LIN {X 0,Y 112.861,Z 852.907,A -85,B 0,C 180,E1 29250,E2 29250} C_VEL
LIN {X 0,Y 107.228,Z 852.568,A -85,B 0,C 180,E1 29258.656,E2 29258.656} C_VEL
LIN {X 0,Y 96.977,Z 851.298,A -85,B 0,C 180,E1 29270.448,E2 29270.448} C_VEL
LIN {X 0,Y 87.732,Z 849.973,A -85,B 0,C 180,E1 29281.18,E2 29281.18} C_VEL
LIN {X 0,Y 77.61,Z 847.953,A -85,B 0,C 180,E1 29299.217,E2 29299.217} C_VEL
LIN {X 0,Y 60.63,Z 851.717,A -85,B 0,C 180,E1 29291.445,E2 29291.445} C_VEL
LIN {X 0,Y 43.178,Z 854.592,A -85,B 0,C 180,E1 29270.527,E2 29270.527} C_VEL
LIN {X 0,Y 38.153,Z 855.115,A -85,B 0,C 180,E1 29250,E2 29250} C_VEL
LIN {X 0,Y 52.851,Z 853.16,A -85,B 0,C 180,E1 29215.044,E2 29215.044} C_VEL
LIN {X 0,Y 73.881,Z 848.759,A -85,B 0,C 180,E1 29201.493,E2 29201.493} C_VEL
LIN {X 0,Y 77.759,Z 847.956,A -85,B 0,C 180,E1 29200.969,E2 29200.969} C_VEL
LIN {X 0,Y 88.144,Z 850.008,A -85,B 0,C 180,E1 29219.219,E2 29219.219} C_VEL
LIN {X 0,Y 99.484,Z 851.624,A -85,B 0,C 180,E1 29232.279,E2 29232.279} C_VEL
LIN {X 0,Y 103.001,Z 852.093,A -85,B 0,C 180,E1 29236.946,E2 29236.946} C_VEL
LIN {X 0,Y 106.169,Z 852.823,A -85,B 0,C 180,E1 29243.549,E2 29243.549} C_VEL
LIN {X 0,Y 104.929,Z 853.168,A -85,B 0,C 180,E1 29249.273,E2 29249.273} C_VEL
LIN {X 0,Y 104.315,Z 853.157,A -85,B 0,C 180,E1 29250.038,E2 29250.038} C_VEL
LIN {X 0,Y 97.922,Z 852.917,A -85,B 0,C 180,E1 29258.895,E2 29258.895} C_VEL
LIN {X 0,Y 87.911,Z 851.989,A -85,B 0,C 180,E1 29270.148,E2 29270.148} C_VEL
LIN {X 0,Y 73.225,Z 850.209,A -85,B 0,C 180,E1 29290.242,E2 29290.242} C_VEL
LIN {X 0,Y 50.776,Z 854.353,A -85,B 0,C 180,E1 29267.348,E2 29267.348} C_VEL
LIN {X 0,Y 46.131,Z 854.879,A -85,B 0,C 180,E1 29250,E2 29250} C_VEL
LIN {X 0,Y 59.659,Z 852.918,A -85,B 0,C 180,E1 29219.498,E2 29219.498} C_VEL
LIN {X 0,Y 73.337,Z 850.187,A -85,B 0,C 180,E1 29209.732,E2 29209.732} C_VEL
LIN {X 0,Y 87.957,Z 851.988,A -85,B 0,C 180,E1 29229.863,E2 29229.863} C_VEL
LIN {X 0,Y 97.92,Z 852.917,A -85,B 0,C 180,E1 29241.105,E2 29241.105} C_VEL
LIN {X 0,Y 104.315,Z 853.157,A -85,B 0,C 180,E1 29250.038,E2 29250.038} C_VEL
LIN {X 0,Y 96.304,Z 853.179,A -85,B 0,C 180,E1 29256,E2 29256} C_VEL
LIN {X 0,Y 81.253,Z 852.795,A -85,B 0,C 180,E1 29266.922,E2 29266.922} C_VEL
LIN {X 0,Y 70.197,Z 851.958,A -85,B 0,C 180,E1 29280.333,E2 29280.333} C_VEL
LIN {X 0,Y 54.121,Z 854.643,A -85,B 0,C 180,E1 29250,E2 29250} C_VEL
LIN {X 0,Y 70.111,Z 851.984,A -85,B 0,C 180,E1 29219.787,E2 29219.787} C_VEL
LIN {X 0,Y 79.937,Z 852.696,A -85,B 0,C 180,E1 29231.322,E2 29231.322} C_VEL
LIN {X 0,Y 88.018,Z 853.216,A -85,B 0,C 180,E1 29240.095,E2 29240.095} C_VEL
LIN {X 0,Y 95.517,Z 853.419,A -85,B 0,C 180,E1 29250,E2 29250} C_VEL
LIN {X 0,Y 88.015,Z 853.216,A -85,B 0,C 180,E1 29259.905,E2 29259.905} C_VEL
LIN {X 0,Y 81.253,Z 852.795,A -85,B 0,C 180,E1 29266.922,E2 29266.922} C_VEL
LIN {X 0,Y 76.697,Z 852.983,A -85,B 0,C 180,E1 29267.815,E2 29267.815} C_VEL
LIN {X 0,Y 68.723,Z 853.725,A -85,B 0,C 180,E1 29263.696,E2 29263.696} C_VEL
LIN {X 0,Y 63.261,Z 854.209,A -85,B 0,C 180,E1 29255.087,E2 29255.087} C_VEL
LIN {X 0,Y 62.099,Z 854.407,A -85,B 0,C 180,E1 29250,E2 29250} C_VEL
LIN {X 0,Y 67.517,Z 853.655,A -85,B 0,C 180,E1 29234.618,E2 29234.618} C_VEL
LIN {X 0,Y 70.634,Z 853.256,A -85,B 0,C 180,E1 29231.795,E2 29231.795} C_VEL
LIN {X 0,Y 81.708,Z 853.612,A -85,B 0,C 180,E1 29243.461,E2 29243.461} C_VEL
LIN {X 0,Y 86.693,Z 853.68,A -85,B 0,C 180,E1 29250,E2 29250} C_VEL
LIN {X 0,Y 81.704,Z 853.612,A -85,B 0,C 180,E1 29256.541,E2 29256.541} C_VEL
LIN {X 0,Y 70.562,Z 853.261,A -85,B 0,C 180,E1 29268.197,E2 29268.197} C_VEL
LIN {X 0,Y 66.314,Z 853.874,A -85,B 0,C 180,E1 29263.198,E2 29263.198} C_VEL
LIN {X 0,Y 63.261,Z 854.209,A -85,B 0,C 180,E1 29255.087,E2 29255.087} C_VEL
LIN {X 0,Y 64.956,Z 854.291,A -85,B 0,C 180,E1 29248.536,E2 29248.536} C_VEL
LIN {X 0,Y 70.805,Z 854.008,A -85,B 0,C 180,E1 29244.483,E2 29244.483} C_VEL
LIN {X 0,Y 73.194,Z 853.938,A -85,B 0,C 180,E1 29244.98,E2 29244.98} C_VEL
LIN {X 0,Y 77.516,Z 853.951,A -85,B 0,C 180,E1 29250,E2 29250} C_VEL
LIN {X 0,Y 73.194,Z 853.938,A -85,B 0,C 180,E1 29255.016,E2 29255.016} C_VEL
LIN {X 0,Y 70.1,Z 854.17,A -85,B 0,C 180,E1 29250,E2 29250} C_VEL
LIN {X 0,Y 73.194,Z 853.938,A -85,B 0,C 180,E1 29244.98,E2 29244.98} C_VEL
LIN {X 0,Y 74.21,Z 855.937,A -85,B 0,C 180,E1 29243.58,E2 29243.58} C_VEL
LIN {X 0,Y 74.21,Z 875,A -85,B 0,C 180,E1 29243.58,E2 29243.58} C_VEL
LIN {X 0,Y 74.21,Z 875,A -85,B 0,C 180,E1 29243.58,E2 29243.58}

QRS_NEXT_CUT()
PTP {E1 29336.94,E2 29336.94}
PTP {X 0,Y 607.852,A -85,B 0,C 180,E1 29336.94,E2 29336.94,E3 0,E4 0,E5 0,E6 0}
QRS_SPEED_INIT()
LIN {X 0,Y 607.852,Z 875,A -85,B 0,C 180,E1 29336.94,E2 29336.94,E3 0,E4 0,E5 0,E6 0} C_VEL
LIN {X 0,Y 607.852,Z 359.34,A -85,B 0,C 180,E1 29336.94,E2 29336.94} C_VEL
LIN {X 0,Y 607.852,Z 351.263,A -85,B 0,C 180,E1 29336.94,E2 29336.94} C_VEL
LIN {X 0,Y 607.872,Z 349.263,A -85,B 0,C 180,E1 29336.752,E2 29336.752} C_VEL
LIN {X 0,Y 607.835,Z 349.264,A -85,B 0,C 180,E1 29333.582,E2 29333.582} C_VEL
LIN {X 0,Y 607.853,Z 349.263,A -85,B 0,C 180,E1 29330.824,E2 29330.824} C_VEL
LIN {X 0,Y 607.845,Z 349.264,A -85,B 0,C 180,E1 29327.658,E2 29327.658} C_VEL
LIN {X 0,Y 607.838,Z 349.264,A -85,B 0,C 180,E1 29324.918,E2 29324.918} C_VEL
LIN {X 0,Y 607.857,Z 349.264,A -85,B 0,C 180,E1 29321.695,E2 29321.695} C_VEL
LIN {X 0,Y 607.831,Z 349.264,A -85,B 0,C 180,E1 29318.992,E2 29318.992} C_VEL
LIN {X 0,Y 607.895,Z 349.264,A -85,B 0,C 180,E1 29315.899,E2 29315.899} C_VEL
LIN {X 0,Y 607.83,Z 349.264,A -85,B 0,C 180,E1 29312.9,E2 29312.9} C_VEL
LIN {X 0,Y 607.892,Z 349.265,A -85,B 0,C 180,E1 29309.788,E2 29309.788} C_VEL
LIN {X 0,Y 607.829,Z 349.264,A -85,B 0,C 180,E1 29306.852,E2 29306.852} C_VEL
LIN {X 0,Y 607.91,Z 349.265,A -85,B 0,C 180,E1 29303.818,E2 29303.818} C_VEL
LIN {X 0,Y 607.828,Z 349.264,A -85,B 0,C 180,E1 29300.835,E2 29300.835} C_VEL
LIN {X 0,Y 607.916,Z 349.265,A -85,B 0,C 180,E1 29297.734,E2 29297.734} C_VEL
LIN {X 0,Y 607.828,Z 349.265,A -85,B 0,C 180,E1 29294.724,E2 29294.724} C_VEL
LIN {X 0,Y 607.914,Z 349.265,A -85,B 0,C 180,E1 29291.705,E2 29291.705} C_VEL
LIN {X 0,Y 607.827,Z 349.265,A -85,B 0,C 180,E1 29288.626,E2 29288.626} C_VEL
LIN {X 0,Y 607.912,Z 349.265,A -85,B 0,C 180,E1 29285.607,E2 29285.607} C_VEL
LIN {X 0,Y 607.828,Z 349.265,A -85,B 0,C 180,E1 29282.638,E2 29282.638} C_VEL
LIN {X 0,Y 607.88,Z 349.264,A -85,B 0,C 180,E1 29279.734,E2 29279.734} C_VEL
LIN {X 0,Y 607.832,Z 349.265,A -85,B 0,C 180,E1 29276.683,E2 29276.683} C_VEL
LIN {X 0,Y 607.852,Z 349.265,A -85,B 0,C 180,E1 29273.868,E2 29273.868} C_VEL
LIN {X 0,Y 607.834,Z 349.265,A -85,B 0,C 180,E1 29270.636,E2 29270.636} C_VEL
LIN {X 0,Y 607.839,Z 349.265,A -85,B 0,C 180,E1 29267.914,E2 29267.914} C_VEL
LIN {X 0,Y 607.836,Z 349.265,A -85,B 0,C 180,E1 29264.576,E2 29264.576} C_VEL
LIN {X 0,Y 607.835,Z 349.265,A -85,B 0,C 180,E1 29261.865,E2 29261.865} C_VEL
LIN {X 0,Y 607.846,Z 349.265,A -85,B 0,C 180,E1 29258.609,E2 29258.609} C_VEL
LIN {X 0,Y 607.827,Z 349.265,A -85,B 0,C 180,E1 29255.948,E2 29255.948} C_VEL
LIN {X 0,Y 607.897,Z 349.265,A -85,B 0,C 180,E1 29252.923,E2 29252.923} C_VEL
LIN {X 0,Y 607.825,Z 349.265,A -85,B 0,C 180,E1 29249.906,E2 29249.906} C_VEL
LIN {X 0,Y 607.9,Z 349.266,A -85,B 0,C 180,E1 29246.889,E2 29246.889} C_VEL
LIN {X 0,Y 607.825,Z 349.265,A -85,B 0,C 180,E1 29243.957,E2 29243.957} C_VEL
LIN {X 0,Y 607.893,Z 349.265,A -85,B 0,C 180,E1 29241.011,E2 29241.011} C_VEL
LIN {X 0,Y 607.827,Z 349.265,A -85,B 0,C 180,E1 29237.942,E2 29237.942} C_VEL
LIN {X 0,Y 607.875,Z 349.265,A -85,B 0,C 180,E1 29235.035,E2 29235.035} C_VEL
LIN {X 0,Y 607.83,Z 349.265,A -85,B 0,C 180,E1 29231.924,E2 29231.924} C_VEL
LIN {X 0,Y 607.857,Z 349.265,A -85,B 0,C 180,E1 29229.088,E2 29229.088} C_VEL
LIN {X 0,Y 607.834,Z 349.265,A -85,B 0,C 180,E1 29225.897,E2 29225.897} C_VEL
LIN {X 0,Y 607.846,Z 349.265,A -85,B 0,C 180,E1 29223.106,E2 29223.106} C_VEL
LIN {X 0,Y 607.84,Z 349.265,A -85,B 0,C 180,E1 29219.888,E2 29219.888} C_VEL
LIN {X 0,Y 607.838,Z 349.265,A -85,B 0,C 180,E1 29217.125,E2 29217.125} C_VEL
LIN {X 0,Y 607.842,Z 349.264,A -85,B 0,C 180,E1 29213.807,E2 29213.807} C_VEL
LIN {X 0,Y 607.835,Z 349.265,A -85,B 0,C 180,E1 29211.071,E2 29211.071} C_VEL
LIN {X 0,Y 607.855,Z 349.264,A -85,B 0,C 180,E1 29207.848,E2 29207.848} C_VEL
LIN {X 0,Y 607.83,Z 349.265,A -85,B 0,C 180,E1 29205.116,E2 29205.116} C_VEL
LIN {X 0,Y 607.902,Z 349.264,A -85,B 0,C 180,E1 29202.118,E2 29202.118} C_VEL
LIN {X 0,Y 607.829,Z 349.264,A -85,B 0,C 180,E1 29199.068,E2 29199.068} C_VEL
LIN {X 0,Y 607.913,Z 349.264,A -85,B 0,C 180,E1 29196.065,E2 29196.065} C_VEL
LIN {X 0,Y 607.829,Z 349.264,A -85,B 0,C 180,E1 29193.094,E2 29193.094} C_VEL
LIN {X 0,Y 607.908,Z 349.265,A -85,B 0,C 180,E1 29190.102,E2 29190.102} C_VEL
LIN {X 0,Y 607.83,Z 349.264,A -85,B 0,C 180,E1 29187.1,E2 29187.1} C_VEL
LIN {X 0,Y 607.9,Z 349.264,A -85,B 0,C 180,E1 29184.067,E2 29184.067} C_VEL
LIN {X 0,Y 607.831,Z 349.264,A -85,B 0,C 180,E1 29181.008,E2 29181.008} C_VEL
LIN {X 0,Y 607.867,Z 349.264,A -85,B 0,C 180,E1 29178.206,E2 29178.206} C_VEL
LIN {X 0,Y 607.836,Z 349.264,A -85,B 0,C 180,E1 29175.059,E2 29175.059} C_VEL
LIN {X 0,Y 607.845,Z 349.264,A -85,B 0,C 180,E1 29172.342,E2 29172.342} C_VEL
LIN {X 0,Y 607.845,Z 349.263,A -85,B 0,C 180,E1 29169.081,E2 29169.081} C_VEL
LIN {X 0,Y 607.835,Z 349.264,A -85,B 0,C 180,E1 29166.418,E2 29166.418} C_VEL
LIN {X 0,Y 607.872,Z 349.263,A -85,B 0,C 180,E1 29163.248,E2 29163.248} C_VEL
LIN {X 0,Y 607.833,Z 349.264,A -85,B 0,C 180,E1 29160.373,E2 29160.373} C_VEL
LIN {X 0,Y 607.888,Z 349.263,A -85,B 0,C 180,E1 29157.262,E2 29157.262} C_VEL
LIN {X 0,Y 607.833,Z 349.263,A -85,B 0,C 180,E1 29154.332,E2 29154.332} C_VEL
LIN {X 0,Y 607.904,Z 349.264,A -85,B 0,C 180,E1 29151.292,E2 29151.292} C_VEL
LIN {X 0,Y 607.832,Z 349.264,A -85,B 0,C 180,E1 29148.323,E2 29148.323} C_VEL
LIN {X 0,Y 607.915,Z 349.264,A -85,B 0,C 180,E1 29145.325,E2 29145.325} C_VEL
LIN {X 0,Y 607.832,Z 349.264,A -85,B 0,C 180,E1 29142.251,E2 29142.251} C_VEL
LIN {X 0,Y 607.909,Z 349.264,A -85,B 0,C 180,E1 29139.187,E2 29139.187} C_VEL
LIN {X 0,Y 607.833,Z 349.264,A -85,B 0,C 180,E1 29136.128,E2 29136.128} C_VEL
LIN {X 0,Y 607.911,Z 349.264,A -85,B 0,C 180,E1 29133.106,E2 29133.106} C_VEL
LIN {X 0,Y 607.834,Z 349.264,A -85,B 0,C 180,E1 29130.096,E2 29130.096} C_VEL
LIN {X 0,Y 607.907,Z 349.265,A -85,B 0,C 180,E1 29127.125,E2 29127.125} C_VEL
LIN {X 0,Y 607.838,Z 349.264,A -85,B 0,C 180,E1 29124.153,E2 29124.153} C_VEL
LIN {X 0,Y 607.861,Z 349.264,A -85,B 0,C 180,E1 29121.379,E2 29121.379} C_VEL
LIN {X 0,Y 607.844,Z 349.263,A -85,B 0,C 180,E1 29118.17,E2 29118.17} C_VEL
LIN {X 0,Y 607.852,Z 349.264,A -85,B 0,C 180,E1 29115.381,E2 29115.381} C_VEL
LIN {X 0,Y 607.846,Z 349.263,A -85,B 0,C 180,E1 29112.109,E2 29112.109} C_VEL
LIN {X 0,Y 607.847,Z 349.264,A -85,B 0,C 180,E1 29109.364,E2 29109.364} C_VEL
LIN {X 0,Y 607.852,Z 349.263,A -85,B 0,C 180,E1 29106.076,E2 29106.076} C_VEL
LIN {X 0,Y 607.844,Z 349.263,A -85,B 0,C 180,E1 29103.318,E2 29103.318} C_VEL
LIN {X 0,Y 607.896,Z 349.549,A -85,B 0,C 180,E1 29102.807,E2 29102.807} C_VEL
LIN {X 0,Y 607.904,Z 374.795,A -85,B 0,C 180,E1 29099.891,E2 29099.891} C_VEL
LIN {X 0,Y 607.881,Z 395.066,A -85,B 0,C 180,E1 29097.648,E2 29097.648} C_VEL
LIN {X 0,Y 607.918,Z 609.038,A -85,B 0,C 180,E1 29094.874,E2 29094.874} C_VEL
LIN {X 0,Y 607.917,Z 654.447,A -85,B 0,C 180,E1 29094.265,E2 29094.265} C_VEL
LIN {X 0,Y 607.906,Z 675.785,A -85,B 0,C 180,E1 29093.789,E2 29093.789} C_VEL
LIN {X 0,Y 607.91,Z 694.347,A -85,B 0,C 180,E1 29093.204,E2 29093.204} C_VEL
LIN {X 0,Y 607.913,Z 713.651,A -85,B 0,C 180,E1 29092.43,E2 29092.43} C_VEL
LIN {X 0,Y 607.919,Z 732.066,A -85,B 0,C 180,E1 29091.516,E2 29091.516} C_VEL
LIN {X 0,Y 607.917,Z 750.545,A -85,B 0,C 180,E1 29090.406,E2 29090.406} C_VEL
LIN {X 0,Y 607.912,Z 768.568,A -85,B 0,C 180,E1 29089.105,E2 29089.105} C_VEL
LIN {X 0,Y 607.916,Z 785.369,A -85,B 0,C 180,E1 29087.665,E2 29087.665} C_VEL
LIN {X 0,Y 607.909,Z 800.458,A -85,B 0,C 180,E1 29086.138,E2 29086.138} C_VEL
LIN {X 0,Y 607.911,Z 813.589,A -85,B 0,C 180,E1 29084.574,E2 29084.574} C_VEL
LIN {X 0,Y 607.917,Z 825.378,A -85,B 0,C 180,E1 29082.925,E2 29082.925} C_VEL
LIN {X 0,Y 607.912,Z 836.326,A -85,B 0,C 180,E1 29081.095,E2 29081.095} C_VEL
LIN {X 0,Y 607.917,Z 845.249,A -85,B 0,C 180,E1 29079.275,E2 29079.275} C_VEL
LIN {X 0,Y 607.914,Z 852.378,A -85,B 0,C 180,E1 29077.466,E2 29077.466} C_VEL
LIN {X 0,Y 607.912,Z 858.002,A -85,B 0,C 180,E1 29075.569,E2 29075.569} C_VEL
LIN {X 0,Y 607.911,Z 861.924,A -85,B 0,C 180,E1 29073.678,E2 29073.678} C_VEL
LIN {X 0,Y 607.907,Z 864.307,A -85,B 0,C 180,E1 29071.696,E2 29071.696} C_VEL
LIN {X 0,Y 607.907,Z 864.962,A -85,B 0,C 180,E1 29069.812,E2 29069.812} C_VEL
LIN {X 0,Y 607.909,Z 863.95,A -85,B 0,C 180,E1 29067.832,E2 29067.832} C_VEL
LIN {X 0,Y 607.909,Z 861.135,A -85,B 0,C 180,E1 29065.85,E2 29065.85} C_VEL
LIN {X 0,Y 607.916,Z 856.736,A -85,B 0,C 180,E1 29063.958,E2 29063.958} C_VEL
LIN {X 0,Y 607.905,Z 850.621,A -85,B 0,C 180,E1 29062.059,E2 29062.059} C_VEL
LIN {X 0,Y 607.903,Z 843.098,A -85,B 0,C 180,E1 29060.247,E2 29060.247} C_VEL
LIN {X 0,Y 607.904,Z 833.718,A -85,B 0,C 180,E1 29058.425,E2 29058.425} C_VEL
LIN {X 0,Y 607.915,Z 822.179,A -85,B 0,C 180,E1 29056.591,E2 29056.591} C_VEL
LIN {X 0,Y 607.917,Z 809.38,A -85,B 0,C 180,E1 29054.897,E2 29054.897} C_VEL
LIN {X 0,Y 607.911,Z 795.823,A -85,B 0,C 180,E1 29053.371,E2 29053.371} C_VEL
LIN {X 0,Y 607.912,Z 780.817,A -85,B 0,C 180,E1 29051.927,E2 29051.927} C_VEL
LIN {X 0,Y 607.916,Z 763.955,A -85,B 0,C 180,E1 29050.546,E2 29050.546} C_VEL
LIN {X 0,Y 607.918,Z 746.338,A -85,B 0,C 180,E1 29049.329,E2 29049.329} C_VEL
LIN {X 0,Y 607.918,Z 728.275,A -85,B 0,C 180,E1 29048.281,E2 29048.281} C_VEL
LIN {X 0,Y 607.918,Z 709.066,A -85,B 0,C 180,E1 29047.365,E2 29047.365} C_VEL
LIN {X 0,Y 607.916,Z 690.111,A -85,B 0,C 180,E1 29046.649,E2 29046.649} C_VEL
LIN {X 0,Y 607.907,Z 670.6,A -85,B 0,C 180,E1 29046.082,E2 29046.082} C_VEL
LIN {X 0,Y 607.917,Z 650.327,A -85,B 0,C 180,E1 29045.67,E2 29045.67} C_VEL
LIN {X 0,Y 607.884,Z 404.447,A -85,B 0,C 180,E1 29042.485,E2 29042.485} C_VEL
LIN {X 0,Y 607.881,Z 394.817,A -85,B 0,C 180,E1 29042.339,E2 29042.339} C_VEL
LIN {X 0,Y 607.916,Z 367.575,A -85,B 0,C 180,E1 29039.288,E2 29039.288} C_VEL
LIN {X 0,Y 607.891,Z 349.374,A -85,B 0,C 180,E1 29037.152,E2 29037.152} C_VEL
LIN {X 0,Y 607.836,Z 349.264,A -85,B 0,C 180,E1 29034.272,E2 29034.272} C_VEL
LIN {X 0,Y 607.913,Z 349.265,A -85,B 0,C 180,E1 29031.198,E2 29031.198} C_VEL
LIN {X 0,Y 607.835,Z 349.263,A -85,B 0,C 180,E1 29028.227,E2 29028.227} C_VEL
LIN {X 0,Y 607.914,Z 349.263,A -85,B 0,C 180,E1 29025.257,E2 29025.257} C_VEL
LIN {X 0,Y 607.835,Z 349.264,A -85,B 0,C 180,E1 29022.251,E2 29022.251} C_VEL
LIN {X 0,Y 607.885,Z 349.263,A -85,B 0,C 180,E1 29019.372,E2 29019.372} C_VEL
LIN {X 0,Y 607.839,Z 349.264,A -85,B 0,C 180,E1 29016.294,E2 29016.294} C_VEL
LIN {X 0,Y 607.853,Z 349.263,A -85,B 0,C 180,E1 29013.554,E2 29013.554} C_VEL
LIN {X 0,Y 607.844,Z 349.264,A -85,B 0,C 180,E1 29010.281,E2 29010.281} C_VEL
LIN {X 0,Y 607.855,Z 349.262,A -85,B 0,C 180,E1 29007.426,E2 29007.426} C_VEL
LIN {X 0,Y 607.843,Z 349.264,A -85,B 0,C 180,E1 29004.182,E2 29004.182} C_VEL
LIN {X 0,Y 607.848,Z 349.263,A -85,B 0,C 180,E1 29001.41,E2 29001.41} C_VEL
LIN {X 0,Y 607.844,Z 349.264,A -85,B 0,C 180,E1 28998.116,E2 28998.116} C_VEL
LIN {X 0,Y 607.844,Z 349.263,A -85,B 0,C 180,E1 28995.36,E2 28995.36} C_VEL
LIN {X 0,Y 607.848,Z 349.264,A -85,B 0,C 180,E1 28992.061,E2 28992.061} C_VEL
LIN {X 0,Y 607.842,Z 349.264,A -85,B 0,C 180,E1 28989.28,E2 28989.28} C_VEL
LIN {X 0,Y 607.846,Z 349.264,A -85,B 0,C 180,E1 28985.952,E2 28985.952} C_VEL
LIN {X 0,Y 607.846,Z 349.264,A -85,B 0,C 180,E1 28983.116,E2 28983.116} C_VEL
LIN {X 0,Y 607.843,Z 349.264,A -85,B 0,C 180,E1 28979.816,E2 28979.816} C_VEL
LIN {X 0,Y 607.842,Z 349.263,A -85,B 0,C 180,E1 28977.081,E2 28977.081} C_VEL
LIN {X 0,Y 607.872,Z 349.263,A -85,B 0,C 180,E1 28976.752,E2 28976.752} C_VEL
LIN {X 0,Y 606.937,Z 349.386,A -85,B 0,C 180,E1 28976.025,E2 28976.025} C_VEL
LIN {X 0,Y 600.442,Z 350.191,A -85,B 0,C 180,E1 28973.989,E2 28973.989} C_VEL
LIN {X 0,Y 599.893,Z 350.253,A -85,B 0,C 180,E1 28973.458,E2 28973.458} C_VEL
LIN {X 0,Y 599.939,Z 350.25,A -85,B 0,C 180,E1 28970.605,E2 28970.605} C_VEL
LIN {X 0,Y 599.897,Z 350.253,A -85,B 0,C 180,E1 28967.491,E2 28967.491} C_VEL
LIN {X 0,Y 599.912,Z 350.253,A -85,B 0,C 180,E1 28964.737,E2 28964.737} C_VEL
LIN {X 0,Y 599.899,Z 350.253,A -85,B 0,C 180,E1 28961.443,E2 28961.443} C_VEL
LIN {X 0,Y 599.917,Z 350.253,A -85,B 0,C 180,E1 28958.599,E2 28958.599} C_VEL
LIN {X 0,Y 599.9,Z 350.252,A -85,B 0,C 180,E1 28955.382,E2 28955.382} C_VEL
LIN {X 0,Y 599.915,Z 350.253,A -85,B 0,C 180,E1 28952.512,E2 28952.512} C_VEL
LIN {X 0,Y 599.902,Z 350.254,A -85,B 0,C 180,E1 28949.316,E2 28949.316} C_VEL
LIN {X 0,Y 599.905,Z 350.253,A -85,B 0,C 180,E1 28946.526,E2 28946.526} C_VEL
LIN {X 0,Y 599.904,Z 350.254,A -85,B 0,C 180,E1 28943.257,E2 28943.257} C_VEL
LIN {X 0,Y 599.895,Z 350.253,A -85,B 0,C 180,E1 28940.587,E2 28940.587} C_VEL
LIN {X 0,Y 599.93,Z 350.254,A -85,B 0,C 180,E1 28937.427,E2 28937.427} C_VEL
LIN {X 0,Y 599.891,Z 350.254,A -85,B 0,C 180,E1 28934.561,E2 28934.561} C_VEL
LIN {X 0,Y 599.943,Z 350.254,A -85,B 0,C 180,E1 28931.423,E2 28931.423} C_VEL
LIN {X 0,Y 599.892,Z 350.254,A -85,B 0,C 180,E1 28928.438,E2 28928.438} C_VEL
LIN {X 0,Y 599.933,Z 350.254,A -85,B 0,C 180,E1 28925.263,E2 28925.263} C_VEL
LIN {X 0,Y 599.888,Z 350.254,A -85,B 0,C 180,E1 28922.458,E2 28922.458} C_VEL
LIN {X 0,Y 599.959,Z 350.255,A -85,B 0,C 180,E1 28919.37,E2 28919.37} C_VEL
LIN {X 0,Y 599.888,Z 350.254,A -85,B 0,C 180,E1 28916.424,E2 28916.424} C_VEL
LIN {X 0,Y 599.973,Z 350.254,A -85,B 0,C 180,E1 28913.349,E2 28913.349} C_VEL
LIN {X 0,Y 599.888,Z 350.254,A -85,B 0,C 180,E1 28910.386,E2 28910.386} C_VEL
LIN {X 0,Y 599.962,Z 350.255,A -85,B 0,C 180,E1 28907.356,E2 28907.356} C_VEL
LIN {X 0,Y 599.889,Z 350.254,A -85,B 0,C 180,E1 28904.379,E2 28904.379} C_VEL
LIN {X 0,Y 599.928,Z 350.254,A -85,B 0,C 180,E1 28901.526,E2 28901.526} C_VEL
LIN {X 0,Y 599.894,Z 350.254,A -85,B 0,C 180,E1 28898.434,E2 28898.434} C_VEL
LIN {X 0,Y 599.898,Z 350.254,A -85,B 0,C 180,E1 28895.739,E2 28895.739} C_VEL
LIN {X 0,Y 599.897,Z 350.254,A -85,B 0,C 180,E1 28892.388,E2 28892.388} C_VEL
LIN {X 0,Y 599.899,Z 350.254,A -85,B 0,C 180,E1 28889.618,E2 28889.618} C_VEL
LIN {X 0,Y 599.896,Z 350.254,A -85,B 0,C 180,E1 28886.273,E2 28886.273} C_VEL
LIN {X 0,Y 599.902,Z 350.254,A -85,B 0,C 180,E1 28883.493,E2 28883.493} C_VEL
LIN {X 0,Y 599.9,Z 350.254,A -85,B 0,C 180,E1 28880.212,E2 28880.212} C_VEL
LIN {X 0,Y 599.902,Z 350.254,A -85,B 0,C 180,E1 28877.389,E2 28877.389} C_VEL
LIN {X 0,Y 599.896,Z 350.254,A -85,B 0,C 180,E1 28874.061,E2 28874.061} C_VEL
LIN {X 0,Y 599.908,Z 350.254,A -85,B 0,C 180,E1 28871.237,E2 28871.237} C_VEL
LIN {X 0,Y 599.898,Z 350.254,A -85,B 0,C 180,E1 28867.976,E2 28867.976} C_VEL
LIN {X 0,Y 599.898,Z 350.254,A -85,B 0,C 180,E1 28865.261,E2 28865.261} C_VEL
LIN {X 0,Y 599.904,Z 350.254,A -85,B 0,C 180,E1 28861.966,E2 28861.966} C_VEL
LIN {X 0,Y 599.895,Z 350.254,A -85,B 0,C 180,E1 28859.225,E2 28859.225} C_VEL
LIN {X 0,Y 599.924,Z 350.254,A -85,B 0,C 180,E1 28856.061,E2 28856.061} C_VEL
LIN {X 0,Y 599.891,Z 350.254,A -85,B 0,C 180,E1 28853.249,E2 28853.249} C_VEL
LIN {X 0,Y 599.955,Z 350.253,A -85,B 0,C 180,E1 28850.188,E2 28850.188} C_VEL
LIN {X 0,Y 599.889,Z 350.254,A -85,B 0,C 180,E1 28847.286,E2 28847.286} C_VEL
LIN {X 0,Y 599.974,Z 350.254,A -85,B 0,C 180,E1 28844.228,E2 28844.228} C_VEL
LIN {X 0,Y 599.89,Z 350.254,A -85,B 0,C 180,E1 28841.264,E2 28841.264} C_VEL
LIN {X 0,Y 599.976,Z 350.253,A -85,B 0,C 180,E1 28838.135,E2 28838.135} C_VEL
LIN {X 0,Y 599.89,Z 350.254,A -85,B 0,C 180,E1 28835.081,E2 28835.081} C_VEL
LIN {X 0,Y 599.971,Z 350.253,A -85,B 0,C 180,E1 28831.995,E2 28831.995} C_VEL
LIN {X 0,Y 599.891,Z 350.253,A -85,B 0,C 180,E1 28828.954,E2 28828.954} C_VEL
LIN {X 0,Y 599.963,Z 350.252,A -85,B 0,C 180,E1 28825.855,E2 28825.855} C_VEL
LIN {X 0,Y 599.892,Z 350.252,A -85,B 0,C 180,E1 28822.828,E2 28822.828} C_VEL
LIN {X 0,Y 599.969,Z 350.252,A -85,B 0,C 180,E1 28819.768,E2 28819.768} C_VEL
LIN {X 0,Y 599.892,Z 350.251,A -85,B 0,C 180,E1 28816.753,E2 28816.753} C_VEL
LIN {X 0,Y 599.967,Z 350.253,A -85,B 0,C 180,E1 28813.683,E2 28813.683} C_VEL
LIN {X 0,Y 599.892,Z 350.252,A -85,B 0,C 180,E1 28810.657,E2 28810.657} C_VEL
LIN {X 0,Y 599.967,Z 350.252,A -85,B 0,C 180,E1 28807.561,E2 28807.561} C_VEL
LIN {X 0,Y 599.892,Z 350.253,A -85,B 0,C 180,E1 28804.584,E2 28804.584} C_VEL
LIN {X 0,Y 599.974,Z 350.251,A -85,B 0,C 180,E1 28801.524,E2 28801.524} C_VEL
LIN {X 0,Y 599.894,Z 350.253,A -85,B 0,C 180,E1 28798.468,E2 28798.468} C_VEL
LIN {X 0,Y 599.971,Z 350.251,A -85,B 0,C 180,E1 28795.408,E2 28795.408} C_VEL
LIN {X 0,Y 599.893,Z 350.251,A -85,B 0,C 180,E1 28792.43,E2 28792.43} C_VEL
LIN {X 0,Y 599.973,Z 350.253,A -85,B 0,C 180,E1 28789.336,E2 28789.336} C_VEL
LIN {X 0,Y 599.894,Z 350.251,A -85,B 0,C 180,E1 28786.306,E2 28786.306} C_VEL
LIN {X 0,Y 599.975,Z 350.253,A -85,B 0,C 180,E1 28783.24,E2 28783.24} C_VEL
LIN {X 0,Y 599.894,Z 350.252,A -85,B 0,C 180,E1 28780.221,E2 28780.221} C_VEL
LIN {X 0,Y 599.975,Z 350.253,A -85,B 0,C 180,E1 28777.149,E2 28777.149} C_VEL
LIN {X 0,Y 599.895,Z 350.253,A -85,B 0,C 180,E1 28774.105,E2 28774.105} C_VEL
LIN {X 0,Y 599.969,Z 350.253,A -85,B 0,C 180,E1 28771.033,E2 28771.033} C_VEL
LIN {X 0,Y 599.895,Z 350.253,A -85,B 0,C 180,E1 28767.991,E2 28767.991} C_VEL
LIN {X 0,Y 599.974,Z 350.252,A -85,B 0,C 180,E1 28764.902,E2 28764.902} C_VEL
LIN {X 0,Y 599.896,Z 350.252,A -85,B 0,C 180,E1 28761.875,E2 28761.875} C_VEL
LIN {X 0,Y 599.975,Z 350.252,A -85,B 0,C 180,E1 28758.83,E2 28758.83} C_VEL
LIN {X 0,Y 599.896,Z 350.253,A -85,B 0,C 180,E1 28755.78,E2 28755.78} C_VEL
LIN {X 0,Y 599.969,Z 350.251,A -85,B 0,C 180,E1 28752.697,E2 28752.697} C_VEL
LIN {X 0,Y 599.896,Z 350.253,A -85,B 0,C 180,E1 28749.668,E2 28749.668} C_VEL
LIN {X 0,Y 599.967,Z 350.248,A -85,B 0,C 180,E1 28746.556,E2 28746.556} C_VEL
LIN {X 0,Y 599.897,Z 350.251,A -85,B 0,C 180,E1 28743.554,E2 28743.554} C_VEL
LIN {X 0,Y 599.967,Z 350.601,A -85,B 0,C 180,E1 28743.171,E2 28743.171} C_VEL
LIN {X 0,Y 600.498,Z 353.702,A -85,B 0,C 180,E1 28742.76,E2 28742.76} C_VEL
LIN {X 0,Y 600.384,Z 380.759,A -85,B 0,C 180,E1 28739.619,E2 28739.619} C_VEL
LIN {X 0,Y 600.4,Z 395.214,A -85,B 0,C 180,E1 28738.016,E2 28738.016} C_VEL
LIN {X 0,Y 600.789,Z 398.717,A -85,B 0,C 180,E1 28737.944,E2 28737.944} C_VEL
LIN {X 0,Y 600.637,Z 633.007,A -85,B 0,C 180,E1 28734.887,E2 28734.887} C_VEL
LIN {X 0,Y 600.605,Z 659.013,A -85,B 0,C 180,E1 28734.489,E2 28734.489} C_VEL
LIN {X 0,Y 600.536,Z 679.148,A -85,B 0,C 180,E1 28734.001,E2 28734.001} C_VEL
LIN {X 0,Y 600.481,Z 698.892,A -85,B 0,C 180,E1 28733.346,E2 28733.346} C_VEL
LIN {X 0,Y 600.409,Z 718.115,A -85,B 0,C 180,E1 28732.52,E2 28732.52} C_VEL
LIN {X 0,Y 600.337,Z 736.524,A -85,B 0,C 180,E1 28731.545,E2 28731.545} C_VEL
LIN {X 0,Y 600.252,Z 754.917,A -85,B 0,C 180,E1 28730.373,E2 28730.373} C_VEL
LIN {X 0,Y 600.171,Z 772.231,A -85,B 0,C 180,E1 28729.058,E2 28729.058} C_VEL
LIN {X 0,Y 600.104,Z 788.161,A -85,B 0,C 180,E1 28727.629,E2 28727.629} C_VEL
LIN {X 0,Y 600.043,Z 802.211,A -85,B 0,C 180,E1 28726.157,E2 28726.157} C_VEL
LIN {X 0,Y 600.004,Z 815.856,A -85,B 0,C 180,E1 28724.475,E2 28724.475} C_VEL
LIN {X 0,Y 599.964,Z 827.922,A -85,B 0,C 180,E1 28722.708,E2 28722.708} C_VEL
LIN {X 0,Y 599.935,Z 838.402,A -85,B 0,C 180,E1 28720.855,E2 28720.855} C_VEL
LIN {X 0,Y 599.925,Z 846.876,A -85,B 0,C 180,E1 28719.013,E2 28719.013} C_VEL
LIN {X 0,Y 599.924,Z 853.905,A -85,B 0,C 180,E1 28717.084,E2 28717.084} C_VEL
LIN {X 0,Y 599.914,Z 859.14,A -85,B 0,C 180,E1 28715.163,E2 28715.163} C_VEL
LIN {X 0,Y 599.909,Z 862.704,A -85,B 0,C 180,E1 28713.248,E2 28713.248} C_VEL
LIN {X 0,Y 599.906,Z 864.642,A -85,B 0,C 180,E1 28711.241,E2 28711.241} C_VEL
LIN {X 0,Y 599.903,Z 864.851,A -85,B 0,C 180,E1 28709.332,E2 28709.332} C_VEL
LIN {X 0,Y 599.906,Z 863.395,A -85,B 0,C 180,E1 28707.325,E2 28707.325} C_VEL
LIN {X 0,Y 599.909,Z 860.165,A -85,B 0,C 180,E1 28705.316,E2 28705.316} C_VEL
LIN {X 0,Y 599.916,Z 855.418,A -85,B 0,C 180,E1 28703.397,E2 28703.397} C_VEL
LIN {X 0,Y 599.926,Z 848.855,A -85,B 0,C 180,E1 28701.47,E2 28701.47} C_VEL
LIN {X 0,Y 599.936,Z 840.79,A -85,B 0,C 180,E1 28699.631,E2 28699.631} C_VEL
LIN {X 0,Y 599.959,Z 830.841,A -85,B 0,C 180,E1 28697.781,E2 28697.781} C_VEL
LIN {X 0,Y 599.985,Z 819.387,A -85,B 0,C 180,E1 28696.017,E2 28696.017} C_VEL
LIN {X 0,Y 600.035,Z 806.937,A -85,B 0,C 180,E1 28694.396,E2 28694.396} C_VEL
LIN {X 0,Y 600.093,Z 792.484,A -85,B 0,C 180,E1 28692.798,E2 28692.798} C_VEL
LIN {X 0,Y 600.158,Z 777.054,A -85,B 0,C 180,E1 28691.345,E2 28691.345} C_VEL
LIN {X 0,Y 600.235,Z 759.765,A -85,B 0,C 180,E1 28689.968,E2 28689.968} C_VEL
LIN {X 0,Y 600.302,Z 742.038,A -85,B 0,C 180,E1 28688.781,E2 28688.781} C_VEL
LIN {X 0,Y 600.377,Z 723.017,A -85,B 0,C 180,E1 28687.721,E2 28687.721} C_VEL
LIN {X 0,Y 600.456,Z 703.999,A -85,B 0,C 180,E1 28686.861,E2 28686.861} C_VEL
LIN {X 0,Y 600.532,Z 683.548,A -85,B 0,C 180,E1 28686.132,E2 28686.132} C_VEL
LIN {X 0,Y 600.592,Z 663.682,A -85,B 0,C 180,E1 28685.606,E2 28685.606} C_VEL
LIN {X 0,Y 600.632,Z 642.736,A -85,B 0,C 180,E1 28685.239,E2 28685.239} C_VEL
LIN {X 0,Y 600.785,Z 407.5,A -85,B 0,C 180,E1 28682.173,E2 28682.173} C_VEL
LIN {X 0,Y 600.547,Z 395.894,A -85,B 0,C 180,E1 28682.006,E2 28682.006} C_VEL
LIN {X 0,Y 600.322,Z 393.971,A -85,B 0,C 180,E1 28681.879,E2 28681.879} C_VEL
LIN {X 0,Y 600.448,Z 366.646,A -85,B 0,C 180,E1 28678.756,E2 28678.756} C_VEL
LIN {X 0,Y 600.278,Z 351.784,A -85,B 0,C 180,E1 28676.999,E2 28676.999} C_VEL
LIN {X 0,Y 599.919,Z 350.327,A -85,B 0,C 180,E1 28676.749,E2 28676.749} C_VEL
LIN {X 0,Y 599.913,Z 350.253,A -85,B 0,C 180,E1 28673.935,E2 28673.935} C_VEL
LIN {X 0,Y 599.909,Z 350.253,A -85,B 0,C 180,E1 28670.656,E2 28670.656} C_VEL
LIN {X 0,Y 599.909,Z 350.251,A -85,B 0,C 180,E1 28667.876,E2 28667.876} C_VEL
LIN {X 0,Y 599.909,Z 350.253,A -85,B 0,C 180,E1 28664.563,E2 28664.563} C_VEL
LIN {X 0,Y 599.906,Z 350.252,A -85,B 0,C 180,E1 28661.813,E2 28661.813} C_VEL
LIN {X 0,Y 599.917,Z 350.252,A -85,B 0,C 180,E1 28658.562,E2 28658.562} C_VEL
LIN {X 0,Y 599.901,Z 350.253,A -85,B 0,C 180,E1 28655.806,E2 28655.806} C_VEL
LIN {X 0,Y 599.94,Z 350.253,A -85,B 0,C 180,E1 28652.684,E2 28652.684} C_VEL
LIN {X 0,Y 599.897,Z 350.253,A -85,B 0,C 180,E1 28649.783,E2 28649.783} C_VEL
LIN {X 0,Y 599.947,Z 350.254,A -85,B 0,C 180,E1 28646.638,E2 28646.638} C_VEL
LIN {X 0,Y 599.895,Z 350.253,A -85,B 0,C 180,E1 28643.79,E2 28643.79} C_VEL
LIN {X 0,Y 599.967,Z 350.253,A -85,B 0,C 180,E1 28640.692,E2 28640.692} C_VEL
LIN {X 0,Y 599.894,Z 350.253,A -85,B 0,C 180,E1 28637.662,E2 28637.662} C_VEL
LIN {X 0,Y 599.966,Z 350.251,A -85,B 0,C 180,E1 28634.578,E2 28634.578} C_VEL
LIN {X 0,Y 599.893,Z 350.253,A -85,B 0,C 180,E1 28631.638,E2 28631.638} C_VEL
LIN {X 0,Y 599.973,Z 350.253,A -85,B 0,C 180,E1 28628.533,E2 28628.533} C_VEL
LIN {X 0,Y 599.894,Z 350.251,A -85,B 0,C 180,E1 28625.455,E2 28625.455} C_VEL
LIN {X 0,Y 599.965,Z 350.254,A -85,B 0,C 180,E1 28622.392,E2 28622.392} C_VEL
LIN {X 0,Y 599.891,Z 350.251,A -85,B 0,C 180,E1 28619.431,E2 28619.431} C_VEL
LIN {X 0,Y 599.973,Z 350.253,A -85,B 0,C 180,E1 28616.374,E2 28616.374} C_VEL
LIN {X 0,Y 599.893,Z 350.253,A -85,B 0,C 180,E1 28613.458,E2 28613.458} C_VEL
LIN {X 0,Y 598.922,Z 350.378,A -85,B 0,C 180,E1 28612.723,E2 28612.723} C_VEL
LIN {X 0,Y 592.491,Z 351.185,A -85,B 0,C 180,E1 28610.605,E2 28610.605} C_VEL
LIN {X 0,Y 592.015,Z 351.241,A -85,B 0,C 180,E1 28610.121,E2 28610.121} C_VEL
LIN {X 0,Y 591.955,Z 351.242,A -85,B 0,C 180,E1 28607.122,E2 28607.122} C_VEL
LIN {X 0,Y 592.016,Z 351.239,A -85,B 0,C 180,E1 28604.026,E2 28604.026} C_VEL
LIN {X 0,Y 591.954,Z 351.241,A -85,B 0,C 180,E1 28601.06,E2 28601.06} C_VEL
LIN {X 0,Y 592.025,Z 351.241,A -85,B 0,C 180,E1 28597.986,E2 28597.986} C_VEL
LIN {X 0,Y 591.953,Z 351.24,A -85,B 0,C 180,E1 28594.922,E2 28594.922} C_VEL
LIN {X 0,Y 592.009,Z 351.243,A -85,B 0,C 180,E1 28591.784,E2 28591.784} C_VEL
LIN {X 0,Y 591.953,Z 351.242,A -85,B 0,C 180,E1 28588.886,E2 28588.886} C_VEL
LIN {X 0,Y 592.023,Z 351.243,A -85,B 0,C 180,E1 28585.786,E2 28585.786} C_VEL
LIN {X 0,Y 591.952,Z 351.242,A -85,B 0,C 180,E1 28582.802,E2 28582.802} C_VEL
LIN {X 0,Y 592.024,Z 351.244,A -85,B 0,C 180,E1 28579.76,E2 28579.76} C_VEL
LIN {X 0,Y 591.951,Z 351.243,A -85,B 0,C 180,E1 28576.713,E2 28576.713} C_VEL
LIN {X 0,Y 592.034,Z 351.243,A -85,B 0,C 180,E1 28573.687,E2 28573.687} C_VEL
LIN {X 0,Y 591.95,Z 351.243,A -85,B 0,C 180,E1 28570.688,E2 28570.688} C_VEL
LIN {X 0,Y 592.027,Z 351.244,A -85,B 0,C 180,E1 28567.632,E2 28567.632} C_VEL
LIN {X 0,Y 591.95,Z 351.243,A -85,B 0,C 180,E1 28564.577,E2 28564.577} C_VEL
LIN {X 0,Y 592.027,Z 351.244,A -85,B 0,C 180,E1 28561.488,E2 28561.488} C_VEL
LIN {X 0,Y 591.95,Z 351.243,A -85,B 0,C 180,E1 28558.445,E2 28558.445} C_VEL
LIN {X 0,Y 592.028,Z 351.244,A -85,B 0,C 180,E1 28555.391,E2 28555.391} C_VEL
LIN {X 0,Y 591.949,Z 351.243,A -85,B 0,C 180,E1 28552.336,E2 28552.336} C_VEL
LIN {X 0,Y 592.027,Z 351.244,A -85,B 0,C 180,E1 28549.276,E2 28549.276} C_VEL
LIN {X 0,Y 591.949,Z 351.243,A -85,B 0,C 180,E1 28546.182,E2 28546.182} C_VEL
LIN {X 0,Y 592.018,Z 351.243,A -85,B 0,C 180,E1 28543.08,E2 28543.08} C_VEL
LIN {X 0,Y 591.95,Z 351.243,A -85,B 0,C 180,E1 28540.019,E2 28540.019} C_VEL
LIN {X 0,Y 592.005,Z 351.243,A -85,B 0,C 180,E1 28536.887,E2 28536.887} C_VEL
LIN {X 0,Y 591.95,Z 351.243,A -85,B 0,C 180,E1 28533.874,E2 28533.874} C_VEL
LIN {X 0,Y 591.989,Z 351.243,A -85,B 0,C 180,E1 28530.677,E2 28530.677} C_VEL
LIN {X 0,Y 591.95,Z 351.243,A -85,B 0,C 180,E1 28527.774,E2 28527.774} C_VEL
LIN {X 0,Y 591.989,Z 351.243,A -85,B 0,C 180,E1 28524.573,E2 28524.573} C_VEL
LIN {X 0,Y 591.949,Z 351.243,A -85,B 0,C 180,E1 28521.746,E2 28521.746} C_VEL
LIN {X 0,Y 592.019,Z 351.243,A -85,B 0,C 180,E1 28518.702,E2 28518.702} C_VEL
LIN {X 0,Y 591.948,Z 351.243,A -85,B 0,C 180,E1 28515.724,E2 28515.724} C_VEL
LIN {X 0,Y 592.028,Z 351.244,A -85,B 0,C 180,E1 28512.709,E2 28512.709} C_VEL
LIN {X 0,Y 591.949,Z 351.243,A -85,B 0,C 180,E1 28509.604,E2 28509.604} C_VEL
LIN {X 0,Y 592.019,Z 351.243,A -85,B 0,C 180,E1 28506.511,E2 28506.511} C_VEL
LIN {X 0,Y 591.951,Z 351.243,A -85,B 0,C 180,E1 28503.519,E2 28503.519} C_VEL
LIN {X 0,Y 592.025,Z 351.243,A -85,B 0,C 180,E1 28500.416,E2 28500.416} C_VEL
LIN {X 0,Y 591.95,Z 351.243,A -85,B 0,C 180,E1 28497.398,E2 28497.398} C_VEL
LIN {X 0,Y 592.024,Z 351.243,A -85,B 0,C 180,E1 28494.313,E2 28494.313} C_VEL
LIN {X 0,Y 591.951,Z 351.243,A -85,B 0,C 180,E1 28491.282,E2 28491.282} C_VEL
LIN {X 0,Y 592.011,Z 351.243,A -85,B 0,C 180,E1 28488.132,E2 28488.132} C_VEL
LIN {X 0,Y 591.951,Z 351.243,A -85,B 0,C 180,E1 28485.177,E2 28485.177} C_VEL
LIN {X 0,Y 592.02,Z 351.243,A -85,B 0,C 180,E1 28482.095,E2 28482.095} C_VEL
LIN {X 0,Y 591.953,Z 351.243,A -85,B 0,C 180,E1 28479.017,E2 28479.017} C_VEL
LIN {X 0,Y 592.003,Z 351.242,A -85,B 0,C 180,E1 28475.87,E2 28475.87} C_VEL
LIN {X 0,Y 591.953,Z 351.243,A -85,B 0,C 180,E1 28472.941,E2 28472.941} C_VEL
LIN {X 0,Y 592.02,Z 351.242,A -85,B 0,C 180,E1 28469.875,E2 28469.875} C_VEL
LIN {X 0,Y 591.952,Z 351.243,A -85,B 0,C 180,E1 28466.898,E2 28466.898} C_VEL
LIN {X 0,Y 592.014,Z 351.24,A -85,B 0,C 180,E1 28463.743,E2 28463.743} C_VEL
LIN {X 0,Y 591.953,Z 351.242,A -85,B 0,C 180,E1 28460.769,E2 28460.769} C_VEL
LIN {X 0,Y 592.02,Z 351.238,A -85,B 0,C 180,E1 28457.692,E2 28457.692} C_VEL
LIN {X 0,Y 591.952,Z 351.242,A -85,B 0,C 180,E1 28454.671,E2 28454.671} C_VEL
LIN {X 0,Y 592.022,Z 351.239,A -85,B 0,C 180,E1 28451.589,E2 28451.589} C_VEL
LIN {X 0,Y 591.955,Z 351.239,A -85,B 0,C 180,E1 28448.543,E2 28448.543} C_VEL
LIN {X 0,Y 592.013,Z 351.241,A -85,B 0,C 180,E1 28445.422,E2 28445.422} C_VEL
LIN {X 0,Y 591.956,Z 351.239,A -85,B 0,C 180,E1 28442.416,E2 28442.416} C_VEL
LIN {X 0,Y 591.999,Z 351.241,A -85,B 0,C 180,E1 28439.222,E2 28439.222} C_VEL
LIN {X 0,Y 591.957,Z 351.242,A -85,B 0,C 180,E1 28436.316,E2 28436.316} C_VEL
LIN {X 0,Y 592.011,Z 351.239,A -85,B 0,C 180,E1 28433.207,E2 28433.207} C_VEL
LIN {X 0,Y 591.956,Z 351.242,A -85,B 0,C 180,E1 28430.272,E2 28430.272} C_VEL
LIN {X 0,Y 592.013,Z 351.237,A -85,B 0,C 180,E1 28427.115,E2 28427.115} C_VEL
LIN {X 0,Y 591.955,Z 351.24,A -85,B 0,C 180,E1 28424.217,E2 28424.217} C_VEL
LIN {X 0,Y 592.031,Z 351.241,A -85,B 0,C 180,E1 28421.178,E2 28421.178} C_VEL
LIN {X 0,Y 591.956,Z 351.239,A -85,B 0,C 180,E1 28418.079,E2 28418.079} C_VEL
LIN {X 0,Y 592.028,Z 351.241,A -85,B 0,C 180,E1 28415.023,E2 28415.023} C_VEL
LIN {X 0,Y 591.956,Z 351.238,A -85,B 0,C 180,E1 28411.992,E2 28411.992} C_VEL
LIN {X 0,Y 592.021,Z 351.241,A -85,B 0,C 180,E1 28408.88,E2 28408.88} C_VEL
LIN {X 0,Y 591.958,Z 351.241,A -85,B 0,C 180,E1 28405.855,E2 28405.855} C_VEL
LIN {X 0,Y 592.011,Z 351.239,A -85,B 0,C 180,E1 28402.698,E2 28402.698} C_VEL
LIN {X 0,Y 591.958,Z 351.242,A -85,B 0,C 180,E1 28399.768,E2 28399.768} C_VEL
LIN {X 0,Y 592.026,Z 351.241,A -85,B 0,C 180,E1 28396.709,E2 28396.709} C_VEL
LIN {X 0,Y 591.958,Z 351.243,A -85,B 0,C 180,E1 28393.694,E2 28393.694} C_VEL
LIN {X 0,Y 592.018,Z 351.239,A -85,B 0,C 180,E1 28390.534,E2 28390.534} C_VEL
LIN {X 0,Y 591.96,Z 351.242,A -85,B 0,C 180,E1 28387.57,E2 28387.57} C_VEL
LIN {X 0,Y 592.018,Z 351.238,A -85,B 0,C 180,E1 28384.455,E2 28384.455} C_VEL
LIN {X 0,Y 592.002,Z 351.54,A -85,B 0,C 180,E1 28383.563,E2 28383.563} C_VEL
LIN {X 0,Y 593.081,Z 356.347,A -85,B 0,C 180,E1 28382.905,E2 28382.905} C_VEL
LIN {X 0,Y 592.868,Z 382.945,A -85,B 0,C 180,E1 28379.779,E2 28379.779} C_VEL
LIN {X 0,Y 592.858,Z 395.198,A -85,B 0,C 180,E1 28378.405,E2 28378.405} C_VEL
LIN {X 0,Y 593.718,Z 399.417,A -85,B 0,C 180,E1 28378.297,E2 28378.297} C_VEL
LIN {X 0,Y 593.377,Z 633.668,A -85,B 0,C 180,E1 28375.204,E2 28375.204} C_VEL
LIN {X 0,Y 593.309,Z 659.39,A -85,B 0,C 180,E1 28374.803,E2 28374.803} C_VEL
LIN {X 0,Y 593.182,Z 679.697,A -85,B 0,C 180,E1 28374.301,E2 28374.301} C_VEL
LIN {X 0,Y 593.05,Z 700.181,A -85,B 0,C 180,E1 28373.603,E2 28373.603} C_VEL
LIN {X 0,Y 592.913,Z 719.242,A -85,B 0,C 180,E1 28372.766,E2 28372.766} C_VEL
LIN {X 0,Y 592.765,Z 737.419,A -85,B 0,C 180,E1 28371.782,E2 28371.782} C_VEL
LIN {X 0,Y 592.595,Z 755.647,A -85,B 0,C 180,E1 28370.596,E2 28370.596} C_VEL
LIN {X 0,Y 592.433,Z 772.839,A -85,B 0,C 180,E1 28369.265,E2 28369.265} C_VEL
LIN {X 0,Y 592.292,Z 789.452,A -85,B 0,C 180,E1 28367.74,E2 28367.74} C_VEL
LIN {X 0,Y 592.171,Z 804.484,A -85,B 0,C 180,E1 28366.108,E2 28366.108} C_VEL
LIN {X 0,Y 592.08,Z 817.975,A -85,B 0,C 180,E1 28364.373,E2 28364.373} C_VEL
LIN {X 0,Y 592.009,Z 829.113,A -85,B 0,C 180,E1 28362.683,E2 28362.683} C_VEL
LIN {X 0,Y 591.961,Z 839.4,A -85,B 0,C 180,E1 28360.806,E2 28360.806} C_VEL
LIN {X 0,Y 591.938,Z 847.69,A -85,B 0,C 180,E1 28358.94,E2 28358.94} C_VEL
LIN {X 0,Y 591.926,Z 854.514,A -85,B 0,C 180,E1 28356.985,E2 28356.985} C_VEL
LIN {X 0,Y 591.919,Z 859.548,A -85,B 0,C 180,E1 28355.039,E2 28355.039} C_VEL
LIN {X 0,Y 591.913,Z 862.951,A -85,B 0,C 180,E1 28353.099,E2 28353.099} C_VEL
LIN {X 0,Y 591.913,Z 864.752,A -85,B 0,C 180,E1 28351.065,E2 28351.065} C_VEL
LIN {X 0,Y 591.916,Z 864.781,A -85,B 0,C 180,E1 28349.032,E2 28349.032} C_VEL
LIN {X 0,Y 591.916,Z 863.063,A -85,B 0,C 180,E1 28346.998,E2 28346.998} C_VEL
LIN {X 0,Y 591.92,Z 859.753,A -85,B 0,C 180,E1 28345.058,E2 28345.058} C_VEL
LIN {X 0,Y 591.926,Z 854.816,A -85,B 0,C 180,E1 28343.112,E2 28343.112} C_VEL
LIN {X 0,Y 591.937,Z 848.088,A -85,B 0,C 180,E1 28341.158,E2 28341.158} C_VEL
LIN {X 0,Y 591.957,Z 839.864,A -85,B 0,C 180,E1 28339.293,E2 28339.293} C_VEL
LIN {X 0,Y 592.004,Z 829.69,A -85,B 0,C 180,E1 28337.416,E2 28337.416} C_VEL
LIN {X 0,Y 592.074,Z 818.681,A -85,B 0,C 180,E1 28335.727,E2 28335.727} C_VEL
LIN {X 0,Y 592.17,Z 805.611,A -85,B 0,C 180,E1 28334.025,E2 28334.025} C_VEL
LIN {X 0,Y 592.286,Z 790.969,A -85,B 0,C 180,E1 28332.412,E2 28332.412} C_VEL
LIN {X 0,Y 592.424,Z 775.181,A -85,B 0,C 180,E1 28330.933,E2 28330.933} C_VEL
LIN {X 0,Y 592.572,Z 758.888,A -85,B 0,C 180,E1 28329.635,E2 28329.635} C_VEL
LIN {X 0,Y 592.737,Z 740.916,A -85,B 0,C 180,E1 28328.425,E2 28328.425} C_VEL
LIN {X 0,Y 592.888,Z 721.309,A -85,B 0,C 180,E1 28327.335,E2 28327.335} C_VEL
LIN {X 0,Y 593.027,Z 702.308,A -85,B 0,C 180,E1 28326.484,E2 28326.484} C_VEL
LIN {X 0,Y 593.176,Z 681.441,A -85,B 0,C 180,E1 28325.752,E2 28325.752} C_VEL
LIN {X 0,Y 593.306,Z 660.639,A -85,B 0,C 180,E1 28325.223,E2 28325.223} C_VEL
LIN {X 0,Y 593.373,Z 637.304,A -85,B 0,C 180,E1 28324.844,E2 28324.844} C_VEL
LIN {X 0,Y 593.714,Z 402.01,A -85,B 0,C 180,E1 28321.738,E2 28321.738} C_VEL
LIN {X 0,Y 593.427,Z 397.378,A -85,B 0,C 180,E1 28321.661,E2 28321.661} C_VEL
LIN {X 0,Y 592.791,Z 394.485,A -85,B 0,C 180,E1 28321.544,E2 28321.544} C_VEL
LIN {X 0,Y 592.998,Z 367.125,A -85,B 0,C 180,E1 28318.375,E2 28318.375} C_VEL
LIN {X 0,Y 592.885,Z 354.661,A -85,B 0,C 180,E1 28316.881,E2 28316.881} C_VEL
LIN {X 0,Y 591.967,Z 351.309,A -85,B 0,C 180,E1 28316.359,E2 28316.359} C_VEL
LIN {X 0,Y 592.037,Z 351.233,A -85,B 0,C 180,E1 28313.285,E2 28313.285} C_VEL
LIN {X 0,Y 591.958,Z 351.241,A -85,B 0,C 180,E1 28310.198,E2 28310.198} C_VEL
LIN {X 0,Y 592.029,Z 351.243,A -85,B 0,C 180,E1 28307.11,E2 28307.11} C_VEL
LIN {X 0,Y 591.958,Z 351.242,A -85,B 0,C 180,E1 28304.101,E2 28304.101} C_VEL
LIN {X 0,Y 592.019,Z 351.243,A -85,B 0,C 180,E1 28300.944,E2 28300.944} C_VEL
LIN {X 0,Y 591.96,Z 351.24,A -85,B 0,C 180,E1 28297.929,E2 28297.929} C_VEL
LIN {X 0,Y 592.014,Z 351.242,A -85,B 0,C 180,E1 28294.812,E2 28294.812} C_VEL
LIN {X 0,Y 591.959,Z 351.241,A -85,B 0,C 180,E1 28291.805,E2 28291.805} C_VEL
LIN {X 0,Y 592.007,Z 351.239,A -85,B 0,C 180,E1 28288.665,E2 28288.665} C_VEL
LIN {X 0,Y 591.957,Z 351.241,A -85,B 0,C 180,E1 28285.73,E2 28285.73} C_VEL
LIN {X 0,Y 592.004,Z 351.239,A -85,B 0,C 180,E1 28282.547,E2 28282.547} C_VEL
LIN {X 0,Y 591.958,Z 351.24,A -85,B 0,C 180,E1 28279.644,E2 28279.644} C_VEL
LIN {X 0,Y 592.009,Z 351.241,A -85,B 0,C 180,E1 28276.487,E2 28276.487} C_VEL
LIN {X 0,Y 591.956,Z 351.238,A -85,B 0,C 180,E1 28273.582,E2 28273.582} C_VEL
LIN {X 0,Y 592.024,Z 351.243,A -85,B 0,C 180,E1 28270.513,E2 28270.513} C_VEL
LIN {X 0,Y 591.955,Z 351.239,A -85,B 0,C 180,E1 28267.477,E2 28267.477} C_VEL
LIN {X 0,Y 592.018,Z 351.243,A -85,B 0,C 180,E1 28264.363,E2 28264.363} C_VEL
LIN {X 0,Y 591.956,Z 351.242,A -85,B 0,C 180,E1 28261.359,E2 28261.359} C_VEL
LIN {X 0,Y 592.016,Z 351.24,A -85,B 0,C 180,E1 28258.262,E2 28258.262} C_VEL
LIN {X 0,Y 591.956,Z 351.242,A -85,B 0,C 180,E1 28255.257,E2 28255.257} C_VEL
LIN {X 0,Y 592.015,Z 351.239,A -85,B 0,C 180,E1 28252.142,E2 28252.142} C_VEL
LIN {X 0,Y 592.015,Z 351.241,A -85,B 0,C 180,E1 28250.121,E2 28250.121} C_VEL
LIN {X 0,Y 590.954,Z 351.37,A -85,B 0,C 180,E1 28249.376,E2 28249.376} C_VEL
LIN {X 0,Y 584.527,Z 352.168,A -85,B 0,C 180,E1 28247.284,E2 28247.284} C_VEL
LIN {X 0,Y 584.038,Z 352.231,A -85,B 0,C 180,E1 28246.74,E2 28246.74} C_VEL
LIN {X 0,Y 584.022,Z 352.226,A -85,B 0,C 180,E1 28243.477,E2 28243.477} C_VEL
LIN {X 0,Y 584.041,Z 352.229,A -85,B 0,C 180,E1 28240.607,E2 28240.607} C_VEL
LIN {X 0,Y 584.019,Z 352.229,A -85,B 0,C 180,E1 28237.332,E2 28237.332} C_VEL
LIN {X 0,Y 584.059,Z 352.228,A -85,B 0,C 180,E1 28234.341,E2 28234.341} C_VEL
LIN {X 0,Y 584.017,Z 352.231,A -85,B 0,C 180,E1 28231.139,E2 28231.139} C_VEL
LIN {X 0,Y 584.066,Z 352.231,A -85,B 0,C 180,E1 28228.187,E2 28228.187} C_VEL
LIN {X 0,Y 584.014,Z 352.232,A -85,B 0,C 180,E1 28225.011,E2 28225.011} C_VEL
LIN {X 0,Y 584.084,Z 352.231,A -85,B 0,C 180,E1 28221.965,E2 28221.965} C_VEL
LIN {X 0,Y 584.013,Z 352.232,A -85,B 0,C 180,E1 28218.875,E2 28218.875} C_VEL
LIN {X 0,Y 584.089,Z 352.232,A -85,B 0,C 180,E1 28215.826,E2 28215.826} C_VEL
LIN {X 0,Y 584.012,Z 352.232,A -85,B 0,C 180,E1 28212.748,E2 28212.748} C_VEL
LIN {X 0,Y 584.085,Z 352.233,A -85,B 0,C 180,E1 28209.68,E2 28209.68} C_VEL
LIN {X 0,Y 584.012,Z 352.232,A -85,B 0,C 180,E1 28206.568,E2 28206.568} C_VEL
LIN {X 0,Y 584.086,Z 352.233,A -85,B 0,C 180,E1 28203.449,E2 28203.449} C_VEL
LIN {X 0,Y 584.013,Z 352.232,A -85,B 0,C 180,E1 28200.375,E2 28200.375} C_VEL
LIN {X 0,Y 584.064,Z 352.232,A -85,B 0,C 180,E1 28197.198,E2 28197.198} C_VEL
LIN {X 0,Y 584.016,Z 352.232,A -85,B 0,C 180,E1 28194.164,E2 28194.164} C_VEL
LIN {X 0,Y 584.045,Z 352.232,A -85,B 0,C 180,E1 28190.964,E2 28190.964} C_VEL
LIN {X 0,Y 584.016,Z 352.232,A -85,B 0,C 180,E1 28188.051,E2 28188.051} C_VEL
LIN {X 0,Y 584.036,Z 352.233,A -85,B 0,C 180,E1 28184.778,E2 28184.778} C_VEL
LIN {X 0,Y 584.015,Z 352.232,A -85,B 0,C 180,E1 28181.955,E2 28181.955} C_VEL
LIN {X 0,Y 584.035,Z 352.233,A -85,B 0,C 180,E1 28178.665,E2 28178.665} C_VEL
LIN {X 0,Y 584.018,Z 352.232,A -85,B 0,C 180,E1 28175.797,E2 28175.797} C_VEL
LIN {X 0,Y 584.024,Z 352.233,A -85,B 0,C 180,E1 28172.453,E2 28172.453} C_VEL
LIN {X 0,Y 584.023,Z 352.233,A -85,B 0,C 180,E1 28169.608,E2 28169.608} C_VEL
LIN {X 0,Y 584.019,Z 352.232,A -85,B 0,C 180,E1 28166.27,E2 28166.27} C_VEL
LIN {X 0,Y 584.031,Z 352.232,A -85,B 0,C 180,E1 28163.414,E2 28163.414} C_VEL
LIN {X 0,Y 584.018,Z 352.232,A -85,B 0,C 180,E1 28160.143,E2 28160.143} C_VEL
LIN {X 0,Y 584.037,Z 352.232,A -85,B 0,C 180,E1 28157.242,E2 28157.242} C_VEL
LIN {X 0,Y 584.016,Z 352.233,A -85,B 0,C 180,E1 28154,E2 28154} C_VEL
LIN {X 0,Y 584.052,Z 352.232,A -85,B 0,C 180,E1 28151.019,E2 28151.019} C_VEL
LIN {X 0,Y 584.015,Z 352.232,A -85,B 0,C 180,E1 28147.831,E2 28147.831} C_VEL
LIN {X 0,Y 584.058,Z 352.232,A -85,B 0,C 180,E1 28144.878,E2 28144.878} C_VEL
LIN {X 0,Y 584.013,Z 352.232,A -85,B 0,C 180,E1 28141.691,E2 28141.691} C_VEL
LIN {X 0,Y 584.075,Z 352.232,A -85,B 0,C 180,E1 28138.659,E2 28138.659} C_VEL
LIN {X 0,Y 584.013,Z 352.232,A -85,B 0,C 180,E1 28135.596,E2 28135.596} C_VEL
LIN {X 0,Y 584.073,Z 352.232,A -85,B 0,C 180,E1 28132.577,E2 28132.577} C_VEL
LIN {X 0,Y 584.012,Z 352.232,A -85,B 0,C 180,E1 28129.416,E2 28129.416} C_VEL
LIN {X 0,Y 584.087,Z 352.233,A -85,B 0,C 180,E1 28126.382,E2 28126.382} C_VEL
LIN {X 0,Y 584.013,Z 352.232,A -85,B 0,C 180,E1 28123.315,E2 28123.315} C_VEL
LIN {X 0,Y 584.086,Z 352.233,A -85,B 0,C 180,E1 28120.23,E2 28120.23} C_VEL
LIN {X 0,Y 584.013,Z 352.231,A -85,B 0,C 180,E1 28117.174,E2 28117.174} C_VEL
LIN {X 0,Y 584.094,Z 352.232,A -85,B 0,C 180,E1 28114.15,E2 28114.15} C_VEL
LIN {X 0,Y 584.014,Z 352.232,A -85,B 0,C 180,E1 28111.012,E2 28111.012} C_VEL
LIN {X 0,Y 584.093,Z 352.232,A -85,B 0,C 180,E1 28107.961,E2 28107.961} C_VEL
LIN {X 0,Y 584.014,Z 352.229,A -85,B 0,C 180,E1 28104.857,E2 28104.857} C_VEL
LIN {X 0,Y 584.073,Z 352.231,A -85,B 0,C 180,E1 28101.695,E2 28101.695} C_VEL
LIN {X 0,Y 584.017,Z 352.23,A -85,B 0,C 180,E1 28098.666,E2 28098.666} C_VEL
LIN {X 0,Y 584.057,Z 352.23,A -85,B 0,C 180,E1 28095.468,E2 28095.468} C_VEL
LIN {X 0,Y 584.018,Z 352.231,A -85,B 0,C 180,E1 28092.553,E2 28092.553} C_VEL
LIN {X 0,Y 584.055,Z 352.226,A -85,B 0,C 180,E1 28089.355,E2 28089.355} C_VEL
LIN {X 0,Y 584.017,Z 352.231,A -85,B 0,C 180,E1 28086.483,E2 28086.483} C_VEL
LIN {X 0,Y 584.065,Z 352.227,A -85,B 0,C 180,E1 28083.332,E2 28083.332} C_VEL
LIN {X 0,Y 584.017,Z 352.227,A -85,B 0,C 180,E1 28080.388,E2 28080.388} C_VEL
LIN {X 0,Y 584.068,Z 352.23,A -85,B 0,C 180,E1 28077.249,E2 28077.249} C_VEL
LIN {X 0,Y 584.018,Z 352.227,A -85,B 0,C 180,E1 28074.297,E2 28074.297} C_VEL
LIN {X 0,Y 584.067,Z 352.23,A -85,B 0,C 180,E1 28071.133,E2 28071.133} C_VEL
LIN {X 0,Y 584.02,Z 352.231,A -85,B 0,C 180,E1 28068.141,E2 28068.141} C_VEL
LIN {X 0,Y 584.052,Z 352.228,A -85,B 0,C 180,E1 28064.906,E2 28064.906} C_VEL
LIN {X 0,Y 584.02,Z 352.231,A -85,B 0,C 180,E1 28062.048,E2 28062.048} C_VEL
LIN {X 0,Y 584.053,Z 352.226,A -85,B 0,C 180,E1 28058.822,E2 28058.822} C_VEL
LIN {X 0,Y 584.021,Z 352.231,A -85,B 0,C 180,E1 28055.952,E2 28055.952} C_VEL
LIN {X 0,Y 584.062,Z 352.225,A -85,B 0,C 180,E1 28052.799,E2 28052.799} C_VEL
LIN {X 0,Y 584.025,Z 352.231,A -85,B 0,C 180,E1 28049.777,E2 28049.777} C_VEL
LIN {X 0,Y 584.04,Z 352.229,A -85,B 0,C 180,E1 28046.481,E2 28046.481} C_VEL
LIN {X 0,Y 584.026,Z 352.231,A -85,B 0,C 180,E1 28043.673,E2 28043.673} C_VEL
LIN {X 0,Y 584.041,Z 352.231,A -85,B 0,C 180,E1 28040.386,E2 28040.386} C_VEL
LIN {X 0,Y 584.027,Z 352.231,A -85,B 0,C 180,E1 28037.549,E2 28037.549} C_VEL
LIN {X 0,Y 584.032,Z 352.232,A -85,B 0,C 180,E1 28034.168,E2 28034.168} C_VEL
LIN {X 0,Y 584.043,Z 352.228,A -85,B 0,C 180,E1 28031.23,E2 28031.23} C_VEL
LIN {X 0,Y 584.032,Z 352.23,A -85,B 0,C 180,E1 28028.044,E2 28028.044} C_VEL
LIN {X 0,Y 584.047,Z 352.234,A -85,B 0,C 180,E1 28025.113,E2 28025.113} C_VEL
LIN {X 0,Y 584.07,Z 352.504,A -85,B 0,C 180,E1 28023.962,E2 28023.962} C_VEL
LIN {X 0,Y 585.667,Z 359.065,A -85,B 0,C 180,E1 28023.044,E2 28023.044} C_VEL
LIN {X 0,Y 585.353,Z 385.342,A -85,B 0,C 180,E1 28019.918,E2 28019.918} C_VEL
LIN {X 0,Y 585.349,Z 395.215,A -85,B 0,C 180,E1 28018.802,E2 28018.802} C_VEL
LIN {X 0,Y 586.669,Z 401.012,A -85,B 0,C 180,E1 28018.646,E2 28018.646} C_VEL
LIN {X 0,Y 586.133,Z 635.703,A -85,B 0,C 180,E1 28015.51,E2 28015.51} C_VEL
LIN {X 0,Y 586.028,Z 660.352,A -85,B 0,C 180,E1 28015.112,E2 28015.112} C_VEL
LIN {X 0,Y 585.841,Z 681.1,A -85,B 0,C 180,E1 28014.582,E2 28014.582} C_VEL
LIN {X 0,Y 585.631,Z 701.458,A -85,B 0,C 180,E1 28013.867,E2 28013.867} C_VEL
LIN {X 0,Y 585.427,Z 720.234,A -85,B 0,C 180,E1 28013.023,E2 28013.023} C_VEL
LIN {X 0,Y 585.197,Z 739.205,A -85,B 0,C 180,E1 28011.973,E2 28011.973} C_VEL
LIN {X 0,Y 584.942,Z 757.15,A -85,B 0,C 180,E1 28010.77,E2 28010.77} C_VEL
LIN {X 0,Y 584.698,Z 774.199,A -85,B 0,C 180,E1 28009.414,E2 28009.414} C_VEL
LIN {X 0,Y 584.486,Z 790.464,A -85,B 0,C 180,E1 28007.882,E2 28007.882} C_VEL
LIN {X 0,Y 584.305,Z 805.051,A -85,B 0,C 180,E1 28006.263,E2 28006.263} C_VEL
LIN {X 0,Y 584.164,Z 818.681,A -85,B 0,C 180,E1 28004.471,E2 28004.471} C_VEL
LIN {X 0,Y 584.052,Z 830.435,A -85,B 0,C 180,E1 28002.629,E2 28002.629} C_VEL
LIN {X 0,Y 583.982,Z 840.325,A -85,B 0,C 180,E1 28000.755,E2 28000.755} C_VEL
LIN {X 0,Y 583.949,Z 848.479,A -85,B 0,C 180,E1 27998.864,E2 27998.864} C_VEL
LIN {X 0,Y 583.93,Z 855.424,A -85,B 0,C 180,E1 27996.785,E2 27996.785} C_VEL
LIN {X 0,Y 583.918,Z 860.161,A -85,B 0,C 180,E1 27994.813,E2 27994.813} C_VEL
LIN {X 0,Y 583.91,Z 863.401,A -85,B 0,C 180,E1 27992.748,E2 27992.748} C_VEL
LIN {X 0,Y 583.903,Z 864.851,A -85,B 0,C 180,E1 27990.687,E2 27990.687} C_VEL
LIN {X 0,Y 583.905,Z 864.647,A -85,B 0,C 180,E1 27988.724,E2 27988.724} C_VEL
LIN {X 0,Y 583.909,Z 862.695,A -85,B 0,C 180,E1 27986.662,E2 27986.662} C_VEL
LIN {X 0,Y 583.915,Z 859.136,A -85,B 0,C 180,E1 27984.695,E2 27984.695} C_VEL
LIN {X 0,Y 583.931,Z 853.912,A -85,B 0,C 180,E1 27982.721,E2 27982.721} C_VEL
LIN {X 0,Y 583.963,Z 846.878,A -85,B 0,C 180,E1 27980.738,E2 27980.738} C_VEL
LIN {X 0,Y 584.007,Z 838.267,A -85,B 0,C 180,E1 27978.818,E2 27978.818} C_VEL
LIN {X 0,Y 584.089,Z 827.908,A -85,B 0,C 180,E1 27976.941,E2 27976.941} C_VEL
LIN {X 0,Y 584.187,Z 816.563,A -85,B 0,C 180,E1 27975.226,E2 27975.226} C_VEL
LIN {X 0,Y 584.331,Z 803.069,A -85,B 0,C 180,E1 27973.499,E2 27973.499} C_VEL
LIN {X 0,Y 584.51,Z 788.441,A -85,B 0,C 180,E1 27971.913,E2 27971.913} C_VEL
LIN {X 0,Y 584.732,Z 771.638,A -85,B 0,C 180,E1 27970.367,E2 27970.367} C_VEL
LIN {X 0,Y 584.956,Z 754.924,A -85,B 0,C 180,E1 27969.07,E2 27969.07} C_VEL
LIN {X 0,Y 585.223,Z 735.643,A -85,B 0,C 180,E1 27967.817,E2 27967.817} C_VEL
LIN {X 0,Y 585.472,Z 717.016,A -85,B 0,C 180,E1 27966.819,E2 27966.819} C_VEL
LIN {X 0,Y 585.703,Z 697.222,A -85,B 0,C 180,E1 27965.967,E2 27965.967} C_VEL
LIN {X 0,Y 585.87,Z 677.541,A -85,B 0,C 180,E1 27965.312,E2 27965.312} C_VEL
LIN {X 0,Y 586.038,Z 657.107,A -85,B 0,C 180,E1 27964.821,E2 27964.821} C_VEL
LIN {X 0,Y 586.151,Z 627.614,A -85,B 0,C 180,E1 27964.383,E2 27964.383} C_VEL
LIN {X 0,Y 586.652,Z 400.084,A -85,B 0,C 180,E1 27961.34,E2 27961.34} C_VEL
LIN {X 0,Y 585.285,Z 394.674,A -85,B 0,C 180,E1 27961.164,E2 27961.164} C_VEL
LIN {X 0,Y 585.577,Z 366.726,A -85,B 0,C 180,E1 27957.878,E2 27957.878} C_VEL
LIN {X 0,Y 585.506,Z 357.537,A -85,B 0,C 180,E1 27956.76,E2 27956.76} C_VEL
LIN {X 0,Y 584.058,Z 352.416,A -85,B 0,C 180,E1 27956.019,E2 27956.019} C_VEL
LIN {X 0,Y 584.037,Z 352.231,A -85,B 0,C 180,E1 27952.758,E2 27952.758} C_VEL
LIN {X 0,Y 584.03,Z 352.23,A -85,B 0,C 180,E1 27949.932,E2 27949.932} C_VEL
LIN {X 0,Y 584.029,Z 352.232,A -85,B 0,C 180,E1 27946.545,E2 27946.545} C_VEL
LIN {X 0,Y 584.049,Z 352.23,A -85,B 0,C 180,E1 27943.603,E2 27943.603} C_VEL
LIN {X 0,Y 584.025,Z 352.232,A -85,B 0,C 180,E1 27940.375,E2 27940.375} C_VEL
LIN {X 0,Y 584.043,Z 352.228,A -85,B 0,C 180,E1 27937.552,E2 27937.552} C_VEL
LIN {X 0,Y 584.024,Z 352.23,A -85,B 0,C 180,E1 27934.283,E2 27934.283} C_VEL
LIN {X 0,Y 584.065,Z 352.23,A -85,B 0,C 180,E1 27931.248,E2 27931.248} C_VEL
LIN {X 0,Y 584.021,Z 352.226,A -85,B 0,C 180,E1 27928.089,E2 27928.089} C_VEL
LIN {X 0,Y 584.083,Z 352.23,A -85,B 0,C 180,E1 27925.016,E2 27925.016} C_VEL
LIN {X 0,Y 584.017,Z 352.227,A -85,B 0,C 180,E1 27921.891,E2 27921.891} C_VEL
LIN {X 0,Y 584.094,Z 352.23,A -85,B 0,C 180,E1 27918.776,E2 27918.776} C_VEL
LIN {X 0,Y 584.017,Z 352.229,A -85,B 0,C 180,E1 27915.697,E2 27915.697} C_VEL
LIN {X 0,Y 584.088,Z 352.23,A -85,B 0,C 180,E1 27912.56,E2 27912.56} C_VEL
LIN {X 0,Y 584.019,Z 352.231,A -85,B 0,C 180,E1 27909.463,E2 27909.463} C_VEL
LIN {X 0,Y 584.064,Z 352.228,A -85,B 0,C 180,E1 27906.294,E2 27906.294} C_VEL
LIN {X 0,Y 584.019,Z 352.231,A -85,B 0,C 180,E1 27903.341,E2 27903.341} C_VEL
LIN {X 0,Y 584.053,Z 352.228,A -85,B 0,C 180,E1 27900.102,E2 27900.102} C_VEL
LIN {X 0,Y 584.021,Z 352.227,A -85,B 0,C 180,E1 27897.159,E2 27897.159} C_VEL
LIN {X 0,Y 584.042,Z 352.231,A -85,B 0,C 180,E1 27893.912,E2 27893.912} C_VEL
LIN {X 0,Y 584.018,Z 352.226,A -85,B 0,C 180,E1 27891.141,E2 27891.141} C_VEL
LIN {X 0,Y 584.057,Z 352.232,A -85,B 0,C 180,E1 27887.95,E2 27887.95} C_VEL
LIN {X 0,Y 584.038,Z 352.231,A -85,B 0,C 180,E1 27886.74,E2 27886.74} C_VEL
LIN {X 0,Y 583.094,Z 352.354,A -85,B 0,C 180,E1 27885.984,E2 27885.984} C_VEL
LIN {X 0,Y 576.531,Z 353.163,A -85,B 0,C 180,E1 27883.808,E2 27883.808} C_VEL
LIN {X 0,Y 576.077,Z 353.213,A -85,B 0,C 180,E1 27883.311,E2 27883.311} C_VEL
LIN {X 0,Y 576.147,Z 353.218,A -85,B 0,C 180,E1 27880.226,E2 27880.226} C_VEL
LIN {X 0,Y 576.076,Z 353.217,A -85,B 0,C 180,E1 27877.128,E2 27877.128} C_VEL
LIN {X 0,Y 576.148,Z 353.22,A -85,B 0,C 180,E1 27873.963,E2 27873.963} C_VEL
LIN {X 0,Y 576.075,Z 353.221,A -85,B 0,C 180,E1 27870.931,E2 27870.931} C_VEL
LIN {X 0,Y 576.144,Z 353.221,A -85,B 0,C 180,E1 27867.814,E2 27867.814} C_VEL
LIN {X 0,Y 576.075,Z 353.221,A -85,B 0,C 180,E1 27864.822,E2 27864.822} C_VEL
LIN {X 0,Y 576.136,Z 353.221,A -85,B 0,C 180,E1 27861.665,E2 27861.665} C_VEL
LIN {X 0,Y 576.079,Z 353.221,A -85,B 0,C 180,E1 27858.57,E2 27858.57} C_VEL
LIN {X 0,Y 576.108,Z 353.221,A -85,B 0,C 180,E1 27855.351,E2 27855.351} C_VEL
LIN {X 0,Y 576.078,Z 353.221,A -85,B 0,C 180,E1 27852.465,E2 27852.465} C_VEL
LIN {X 0,Y 576.101,Z 353.221,A -85,B 0,C 180,E1 27849.178,E2 27849.178} C_VEL
LIN {X 0,Y 576.087,Z 353.221,A -85,B 0,C 180,E1 27846.204,E2 27846.204} C_VEL
LIN {X 0,Y 576.083,Z 353.221,A -85,B 0,C 180,E1 27842.87,E2 27842.87} C_VEL
LIN {X 0,Y 576.095,Z 353.221,A -85,B 0,C 180,E1 27839.989,E2 27839.989} C_VEL
LIN {X 0,Y 576.079,Z 353.222,A -85,B 0,C 180,E1 27836.712,E2 27836.712} C_VEL
LIN {X 0,Y 576.11,Z 353.221,A -85,B 0,C 180,E1 27833.743,E2 27833.743} C_VEL
LIN {X 0,Y 576.075,Z 353.221,A -85,B 0,C 180,E1 27830.523,E2 27830.523} C_VEL
LIN {X 0,Y 576.131,Z 353.221,A -85,B 0,C 180,E1 27827.471,E2 27827.471} C_VEL
LIN {X 0,Y 576.073,Z 353.222,A -85,B 0,C 180,E1 27824.37,E2 27824.37} C_VEL
LIN {X 0,Y 576.138,Z 353.221,A -85,B 0,C 180,E1 27821.309,E2 27821.309} C_VEL
LIN {X 0,Y 576.071,Z 353.222,A -85,B 0,C 180,E1 27818.182,E2 27818.182} C_VEL
LIN {X 0,Y 576.148,Z 353.222,A -85,B 0,C 180,E1 27815.078,E2 27815.078} C_VEL
LIN {X 0,Y 576.071,Z 353.222,A -85,B 0,C 180,E1 27811.989,E2 27811.989} C_VEL
LIN {X 0,Y 576.132,Z 353.222,A -85,B 0,C 180,E1 27808.807,E2 27808.807} C_VEL
LIN {X 0,Y 576.075,Z 353.221,A -85,B 0,C 180,E1 27805.72,E2 27805.72} C_VEL
LIN {X 0,Y 576.097,Z 353.222,A -85,B 0,C 180,E1 27802.421,E2 27802.421} C_VEL
LIN {X 0,Y 576.076,Z 353.222,A -85,B 0,C 180,E1 27799.601,E2 27799.601} C_VEL
LIN {X 0,Y 576.101,Z 353.222,A -85,B 0,C 180,E1 27796.348,E2 27796.348} C_VEL
LIN {X 0,Y 576.078,Z 353.222,A -85,B 0,C 180,E1 27793.463,E2 27793.463} C_VEL
LIN {X 0,Y 576.088,Z 353.221,A -85,B 0,C 180,E1 27790.113,E2 27790.113} C_VEL
LIN {X 0,Y 576.086,Z 353.222,A -85,B 0,C 180,E1 27787.23,E2 27787.23} C_VEL
LIN {X 0,Y 576.085,Z 353.221,A -85,B 0,C 180,E1 27783.954,E2 27783.954} C_VEL
LIN {X 0,Y 576.096,Z 353.221,A -85,B 0,C 180,E1 27781.039,E2 27781.039} C_VEL
LIN {X 0,Y 576.083,Z 353.221,A -85,B 0,C 180,E1 27777.804,E2 27777.804} C_VEL
LIN {X 0,Y 576.108,Z 353.221,A -85,B 0,C 180,E1 27774.816,E2 27774.816} C_VEL
LIN {X 0,Y 576.077,Z 353.221,A -85,B 0,C 180,E1 27771.586,E2 27771.586} C_VEL
LIN {X 0,Y 576.139,Z 353.221,A -85,B 0,C 180,E1 27768.477,E2 27768.477} C_VEL
LIN {X 0,Y 576.074,Z 353.221,A -85,B 0,C 180,E1 27765.339,E2 27765.339} C_VEL
LIN {X 0,Y 576.149,Z 353.221,A -85,B 0,C 180,E1 27762.316,E2 27762.316} C_VEL
LIN {X 0,Y 576.074,Z 353.221,A -85,B 0,C 180,E1 27759.122,E2 27759.122} C_VEL
LIN {X 0,Y 576.147,Z 353.221,A -85,B 0,C 180,E1 27756.029,E2 27756.029} C_VEL
LIN {X 0,Y 576.076,Z 353.221,A -85,B 0,C 180,E1 27753.016,E2 27753.016} C_VEL
LIN {X 0,Y 576.139,Z 353.22,A -85,B 0,C 180,E1 27749.865,E2 27749.865} C_VEL
LIN {X 0,Y 576.077,Z 353.221,A -85,B 0,C 180,E1 27746.818,E2 27746.818} C_VEL
LIN {X 0,Y 576.118,Z 353.217,A -85,B 0,C 180,E1 27743.606,E2 27743.606} C_VEL
LIN {X 0,Y 576.082,Z 353.221,A -85,B 0,C 180,E1 27740.624,E2 27740.624} C_VEL
LIN {X 0,Y 576.101,Z 353.212,A -85,B 0,C 180,E1 27737.345,E2 27737.345} C_VEL
LIN {X 0,Y 576.085,Z 353.22,A -85,B 0,C 180,E1 27734.433,E2 27734.433} C_VEL
LIN {X 0,Y 576.089,Z 353.216,A -85,B 0,C 180,E1 27731.102,E2 27731.102} C_VEL
LIN {X 0,Y 576.099,Z 353.215,A -85,B 0,C 180,E1 27728.177,E2 27728.177} C_VEL
LIN {X 0,Y 576.083,Z 353.22,A -85,B 0,C 180,E1 27724.874,E2 27724.874} C_VEL
LIN {X 0,Y 576.119,Z 353.216,A -85,B 0,C 180,E1 27721.885,E2 27721.885} C_VEL
LIN {X 0,Y 576.081,Z 353.219,A -85,B 0,C 180,E1 27718.703,E2 27718.703} C_VEL
LIN {X 0,Y 576.141,Z 353.221,A -85,B 0,C 180,E1 27715.617,E2 27715.617} C_VEL
LIN {X 0,Y 576.078,Z 353.216,A -85,B 0,C 180,E1 27712.517,E2 27712.517} C_VEL
LIN {X 0,Y 576.152,Z 353.221,A -85,B 0,C 180,E1 27709.396,E2 27709.396} C_VEL
LIN {X 0,Y 576.079,Z 353.214,A -85,B 0,C 180,E1 27706.241,E2 27706.241} C_VEL
LIN {X 0,Y 576.133,Z 353.22,A -85,B 0,C 180,E1 27703.045,E2 27703.045} C_VEL
LIN {X 0,Y 576.083,Z 353.218,A -85,B 0,C 180,E1 27700.003,E2 27700.003} C_VEL
LIN {X 0,Y 576.115,Z 353.219,A -85,B 0,C 180,E1 27696.796,E2 27696.796} C_VEL
LIN {X 0,Y 576.088,Z 353.22,A -85,B 0,C 180,E1 27693.802,E2 27693.802} C_VEL
LIN {X 0,Y 576.09,Z 353.219,A -85,B 0,C 180,E1 27690.401,E2 27690.401} C_VEL
LIN {X 0,Y 576.108,Z 353.22,A -85,B 0,C 180,E1 27687.449,E2 27687.449} C_VEL
LIN {X 0,Y 576.085,Z 353.22,A -85,B 0,C 180,E1 27684.202,E2 27684.202} C_VEL
LIN {X 0,Y 576.126,Z 353.218,A -85,B 0,C 180,E1 27681.188,E2 27681.188} C_VEL
LIN {X 0,Y 576.084,Z 353.219,A -85,B 0,C 180,E1 27678.069,E2 27678.069} C_VEL
LIN {X 0,Y 576.131,Z 353.22,A -85,B 0,C 180,E1 27675.06,E2 27675.06} C_VEL
LIN {X 0,Y 576.081,Z 353.215,A -85,B 0,C 180,E1 27671.875,E2 27671.875} C_VEL
LIN {X 0,Y 576.157,Z 353.221,A -85,B 0,C 180,E1 27668.789,E2 27668.789} C_VEL
LIN {X 0,Y 576.081,Z 353.217,A -85,B 0,C 180,E1 27665.672,E2 27665.672} C_VEL
LIN {X 0,Y 576.169,Z 353.492,A -85,B 0,C 180,E1 27664.369,E2 27664.369} C_VEL
LIN {X 0,Y 578.256,Z 361.784,A -85,B 0,C 180,E1 27663.186,E2 27663.186} C_VEL
LIN {X 0,Y 577.831,Z 388.218,A -85,B 0,C 180,E1 27660.004,E2 27660.004} C_VEL
LIN {X 0,Y 577.823,Z 395.127,A -85,B 0,C 180,E1 27659.217,E2 27659.217} C_VEL
LIN {X 0,Y 579.64,Z 402.819,A -85,B 0,C 180,E1 27659.001,E2 27659.001} C_VEL
LIN {X 0,Y 578.907,Z 637.964,A -85,B 0,C 180,E1 27655.822,E2 27655.822} C_VEL
LIN {X 0,Y 578.766,Z 661.343,A -85,B 0,C 180,E1 27655.429,E2 27655.429} C_VEL
LIN {X 0,Y 578.517,Z 681.919,A -85,B 0,C 180,E1 27654.889,E2 27654.889} C_VEL
LIN {X 0,Y 578.216,Z 703.233,A -85,B 0,C 180,E1 27654.117,E2 27654.117} C_VEL
LIN {X 0,Y 577.931,Z 722.337,A -85,B 0,C 180,E1 27653.231,E2 27653.231} C_VEL
LIN {X 0,Y 577.604,Z 741.628,A -85,B 0,C 180,E1 27652.122,E2 27652.122} C_VEL
LIN {X 0,Y 577.287,Z 758.515,A -85,B 0,C 180,E1 27650.956,E2 27650.956} C_VEL
LIN {X 0,Y 576.965,Z 775.866,A -85,B 0,C 180,E1 27649.539,E2 27649.539} C_VEL
LIN {X 0,Y 576.681,Z 791.493,A -85,B 0,C 180,E1 27648.025,E2 27648.025} C_VEL
LIN {X 0,Y 576.445,Z 805.619,A -85,B 0,C 180,E1 27646.423,E2 27646.423} C_VEL
LIN {X 0,Y 576.259,Z 818.681,A -85,B 0,C 180,E1 27644.674,E2 27644.674} C_VEL
LIN {X 0,Y 576.114,Z 830.276,A -85,B 0,C 180,E1 27642.835,E2 27642.835} C_VEL
LIN {X 0,Y 576.014,Z 840.322,A -85,B 0,C 180,E1 27640.906,E2 27640.906} C_VEL
LIN {X 0,Y 575.964,Z 848.55,A -85,B 0,C 180,E1 27638.969,E2 27638.969} C_VEL
LIN {X 0,Y 575.936,Z 855.424,A -85,B 0,C 180,E1 27636.88,E2 27636.88} C_VEL
LIN {X 0,Y 575.921,Z 860.16,A -85,B 0,C 180,E1 27634.88,E2 27634.88} C_VEL
LIN {X 0,Y 575.912,Z 863.404,A -85,B 0,C 180,E1 27632.786,E2 27632.786} C_VEL
LIN {X 0,Y 575.904,Z 864.851,A -85,B 0,C 180,E1 27630.696,E2 27630.696} C_VEL
LIN {X 0,Y 575.905,Z 864.65,A -85,B 0,C 180,E1 27628.707,E2 27628.707} C_VEL
LIN {X 0,Y 575.908,Z 862.69,A -85,B 0,C 180,E1 27626.616,E2 27626.616} C_VEL
LIN {X 0,Y 575.917,Z 859.134,A -85,B 0,C 180,E1 27624.621,E2 27624.621} C_VEL
LIN {X 0,Y 575.937,Z 853.915,A -85,B 0,C 180,E1 27622.619,E2 27622.619} C_VEL
LIN {X 0,Y 575.977,Z 846.879,A -85,B 0,C 180,E1 27620.609,E2 27620.609} C_VEL
LIN {X 0,Y 576.043,Z 838.409,A -85,B 0,C 180,E1 27618.689,E2 27618.689} C_VEL
LIN {X 0,Y 576.155,Z 827.902,A -85,B 0,C 180,E1 27616.758,E2 27616.758} C_VEL
LIN {X 0,Y 576.289,Z 816.563,A -85,B 0,C 180,E1 27615.019,E2 27615.019} C_VEL
LIN {X 0,Y 576.505,Z 802.582,A -85,B 0,C 180,E1 27613.209,E2 27613.209} C_VEL
LIN {X 0,Y 576.747,Z 787.936,A -85,B 0,C 180,E1 27611.608,E2 27611.608} C_VEL
LIN {X 0,Y 577.041,Z 771.643,A -85,B 0,C 180,E1 27610.094,E2 27610.094} C_VEL
LIN {X 0,Y 577.339,Z 754.927,A -85,B 0,C 180,E1 27608.78,E2 27608.78} C_VEL
LIN {X 0,Y 577.693,Z 735.648,A -85,B 0,C 180,E1 27607.512,E2 27607.512} C_VEL
LIN {X 0,Y 578.026,Z 716.914,A -85,B 0,C 180,E1 27606.498,E2 27606.498} C_VEL
LIN {X 0,Y 578.342,Z 696.803,A -85,B 0,C 180,E1 27605.626,E2 27605.626} C_VEL
LIN {X 0,Y 578.571,Z 677.4,A -85,B 0,C 180,E1 27604.975,E2 27604.975} C_VEL
LIN {X 0,Y 578.786,Z 656.965,A -85,B 0,C 180,E1 27604.479,E2 27604.479} C_VEL
LIN {X 0,Y 578.94,Z 626.596,A -85,B 0,C 180,E1 27604.026,E2 27604.026} C_VEL
LIN {X 0,Y 579.625,Z 401.816,A -85,B 0,C 180,E1 27600.984,E2 27600.984} C_VEL
LIN {X 0,Y 577.768,Z 394.629,A -85,B 0,C 180,E1 27600.748,E2 27600.748} C_VEL
LIN {X 0,Y 578.169,Z 367.125,A -85,B 0,C 180,E1 27597.465,E2 27597.465} C_VEL
LIN {X 0,Y 578.032,Z 360.059,A -85,B 0,C 180,E1 27596.586,E2 27596.586} C_VEL
LIN {X 0,Y 576.147,Z 353.301,A -85,B 0,C 180,E1 27595.577,E2 27595.577} C_VEL
LIN {X 0,Y 576.084,Z 353.22,A -85,B 0,C 180,E1 27592.47,E2 27592.47} C_VEL
LIN {X 0,Y 576.147,Z 353.209,A -85,B 0,C 180,E1 27589.401,E2 27589.401} C_VEL
LIN {X 0,Y 576.081,Z 353.221,A -85,B 0,C 180,E1 27586.223,E2 27586.223} C_VEL
LIN {X 0,Y 576.152,Z 353.22,A -85,B 0,C 180,E1 27583.065,E2 27583.065} C_VEL
LIN {X 0,Y 576.082,Z 353.22,A -85,B 0,C 180,E1 27580.059,E2 27580.059} C_VEL
LIN {X 0,Y 576.143,Z 353.221,A -85,B 0,C 180,E1 27576.905,E2 27576.905} C_VEL
LIN {X 0,Y 576.082,Z 353.218,A -85,B 0,C 180,E1 27573.86,E2 27573.86} C_VEL
LIN {X 0,Y 576.127,Z 353.22,A -85,B 0,C 180,E1 27570.682,E2 27570.682} C_VEL
LIN {X 0,Y 576.082,Z 353.213,A -85,B 0,C 180,E1 27567.722,E2 27567.722} C_VEL
LIN {X 0,Y 576.117,Z 353.22,A -85,B 0,C 180,E1 27564.509,E2 27564.509} C_VEL
LIN {X 0,Y 576.084,Z 353.214,A -85,B 0,C 180,E1 27561.592,E2 27561.592} C_VEL
LIN {X 0,Y 576.106,Z 353.221,A -85,B 0,C 180,E1 27558.312,E2 27558.312} C_VEL
LIN {X 0,Y 576.086,Z 353.217,A -85,B 0,C 180,E1 27555.403,E2 27555.403} C_VEL
LIN {X 0,Y 576.09,Z 353.22,A -85,B 0,C 180,E1 27552.025,E2 27552.025} C_VEL
LIN {X 0,Y 576.104,Z 353.219,A -85,B 0,C 180,E1 27549.069,E2 27549.069} C_VEL
LIN {X 0,Y 576.087,Z 353.215,A -85,B 0,C 180,E1 27545.881,E2 27545.881} C_VEL
LIN {X 0,Y 576.112,Z 353.219,A -85,B 0,C 180,E1 27542.889,E2 27542.889} C_VEL
LIN {X 0,Y 576.081,Z 353.215,A -85,B 0,C 180,E1 27539.706,E2 27539.706} C_VEL
LIN {X 0,Y 576.12,Z 353.215,A -85,B 0,C 180,E1 27536.715,E2 27536.715} C_VEL
LIN {X 0,Y 576.079,Z 353.22,A -85,B 0,C 180,E1 27533.527,E2 27533.527} C_VEL
LIN {X 0,Y 576.12,Z 353.214,A -85,B 0,C 180,E1 27530.616,E2 27530.616} C_VEL
LIN {X 0,Y 576.08,Z 353.221,A -85,B 0,C 180,E1 27527.475,E2 27527.475} C_VEL
LIN {X 0,Y 576.121,Z 353.219,A -85,B 0,C 180,E1 27524.504,E2 27524.504} C_VEL
LIN {X 0,Y 576.077,Z 353.213,A -85,B 0,C 180,E1 27523.311,E2 27523.311} C_VEL
LIN {X 0,Y 575.098,Z 353.339,A -85,B 0,C 180,E1 27522.545,E2 27522.545} C_VEL
LIN {X 0,Y 568.655,Z 354.156,A -85,B 0,C 180,E1 27520.338,E2 27520.338} C_VEL
LIN {X 0,Y 568.182,Z 354.21,A -85,B 0,C 180,E1 27519.834,E2 27519.834} C_VEL
LIN {X 0,Y 568.145,Z 354.205,A -85,B 0,C 180,E1 27516.79,E2 27516.79} C_VEL
LIN {X 0,Y 568.147,Z 354.21,A -85,B 0,C 180,E1 27513.378,E2 27513.378} C_VEL
LIN {X 0,Y 568.169,Z 354.209,A -85,B 0,C 180,E1 27510.379,E2 27510.379} C_VEL
LIN {X 0,Y 568.142,Z 354.21,A -85,B 0,C 180,E1 27507.185,E2 27507.185} C_VEL
LIN {X 0,Y 568.176,Z 354.21,A -85,B 0,C 180,E1 27504.216,E2 27504.216} C_VEL
LIN {X 0,Y 568.14,Z 354.21,A -85,B 0,C 180,E1 27501.064,E2 27501.064} C_VEL
LIN {X 0,Y 568.194,Z 354.21,A -85,B 0,C 180,E1 27497.951,E2 27497.951} C_VEL
LIN {X 0,Y 568.137,Z 354.21,A -85,B 0,C 180,E1 27494.838,E2 27494.838} C_VEL
LIN {X 0,Y 568.212,Z 354.21,A -85,B 0,C 180,E1 27491.692,E2 27491.692} C_VEL
LIN {X 0,Y 568.135,Z 354.21,A -85,B 0,C 180,E1 27488.534,E2 27488.534} C_VEL
LIN {X 0,Y 568.191,Z 354.211,A -85,B 0,C 180,E1 27485.375,E2 27485.375} C_VEL
LIN {X 0,Y 568.137,Z 354.21,A -85,B 0,C 180,E1 27482.343,E2 27482.343} C_VEL
LIN {X 0,Y 568.165,Z 354.21,A -85,B 0,C 180,E1 27479.058,E2 27479.058} C_VEL
LIN {X 0,Y 568.144,Z 354.211,A -85,B 0,C 180,E1 27476.101,E2 27476.101} C_VEL
LIN {X 0,Y 568.141,Z 354.211,A -85,B 0,C 180,E1 27472.669,E2 27472.669} C_VEL
LIN {X 0,Y 568.165,Z 354.21,A -85,B 0,C 180,E1 27469.721,E2 27469.721} C_VEL
LIN {X 0,Y 568.136,Z 354.211,A -85,B 0,C 180,E1 27466.459,E2 27466.459} C_VEL
LIN {X 0,Y 568.199,Z 354.21,A -85,B 0,C 180,E1 27463.353,E2 27463.353} C_VEL
LIN {X 0,Y 568.134,Z 354.211,A -85,B 0,C 180,E1 27460.136,E2 27460.136} C_VEL
LIN {X 0,Y 568.199,Z 354.211,A -85,B 0,C 180,E1 27456.974,E2 27456.974} C_VEL
LIN {X 0,Y 568.136,Z 354.21,A -85,B 0,C 180,E1 27453.834,E2 27453.834} C_VEL
LIN {X 0,Y 568.154,Z 354.211,A -85,B 0,C 180,E1 27450.504,E2 27450.504} C_VEL
LIN {X 0,Y 568.144,Z 354.211,A -85,B 0,C 180,E1 27447.579,E2 27447.579} C_VEL
LIN {X 0,Y 568.144,Z 354.211,A -85,B 0,C 180,E1 27444.243,E2 27444.243} C_VEL
LIN {X 0,Y 568.161,Z 354.211,A -85,B 0,C 180,E1 27441.295,E2 27441.295} C_VEL
LIN {X 0,Y 568.136,Z 354.21,A -85,B 0,C 180,E1 27438.015,E2 27438.015} C_VEL
LIN {X 0,Y 568.183,Z 354.211,A -85,B 0,C 180,E1 27435.006,E2 27435.006} C_VEL
LIN {X 0,Y 568.136,Z 354.211,A -85,B 0,C 180,E1 27431.841,E2 27431.841} C_VEL
LIN {X 0,Y 568.206,Z 354.21,A -85,B 0,C 180,E1 27428.747,E2 27428.747} C_VEL
LIN {X 0,Y 568.133,Z 354.211,A -85,B 0,C 180,E1 27425.571,E2 27425.571} C_VEL
LIN {X 0,Y 568.204,Z 354.21,A -85,B 0,C 180,E1 27422.433,E2 27422.433} C_VEL
LIN {X 0,Y 568.137,Z 354.21,A -85,B 0,C 180,E1 27419.313,E2 27419.313} C_VEL
LIN {X 0,Y 568.172,Z 354.21,A -85,B 0,C 180,E1 27416.094,E2 27416.094} C_VEL
LIN {X 0,Y 568.142,Z 354.21,A -85,B 0,C 180,E1 27413.123,E2 27413.123} C_VEL
LIN {X 0,Y 568.151,Z 354.21,A -85,B 0,C 180,E1 27409.771,E2 27409.771} C_VEL
LIN {X 0,Y 568.157,Z 354.21,A -85,B 0,C 180,E1 27406.8,E2 27406.8} C_VEL
LIN {X 0,Y 568.141,Z 354.21,A -85,B 0,C 180,E1 27403.471,E2 27403.471} C_VEL
LIN {X 0,Y 568.181,Z 354.21,A -85,B 0,C 180,E1 27400.483,E2 27400.483} C_VEL
LIN {X 0,Y 568.138,Z 354.209,A -85,B 0,C 180,E1 27397.303,E2 27397.303} C_VEL
LIN {X 0,Y 568.206,Z 354.21,A -85,B 0,C 180,E1 27394.206,E2 27394.206} C_VEL
LIN {X 0,Y 568.138,Z 354.21,A -85,B 0,C 180,E1 27391.033,E2 27391.033} C_VEL
LIN {X 0,Y 568.208,Z 354.21,A -85,B 0,C 180,E1 27387.902,E2 27387.902} C_VEL
LIN {X 0,Y 568.139,Z 354.205,A -85,B 0,C 180,E1 27384.755,E2 27384.755} C_VEL
LIN {X 0,Y 568.167,Z 354.209,A -85,B 0,C 180,E1 27381.465,E2 27381.465} C_VEL
LIN {X 0,Y 568.15,Z 354.207,A -85,B 0,C 180,E1 27378.462,E2 27378.462} C_VEL
LIN {X 0,Y 568.145,Z 354.208,A -85,B 0,C 180,E1 27375.092,E2 27375.092} C_VEL
LIN {X 0,Y 568.166,Z 354.21,A -85,B 0,C 180,E1 27372.186,E2 27372.186} C_VEL
LIN {X 0,Y 568.142,Z 354.202,A -85,B 0,C 180,E1 27368.904,E2 27368.904} C_VEL
LIN {X 0,Y 568.177,Z 354.209,A -85,B 0,C 180,E1 27365.955,E2 27365.955} C_VEL
LIN {X 0,Y 568.139,Z 354.203,A -85,B 0,C 180,E1 27362.719,E2 27362.719} C_VEL
LIN {X 0,Y 568.214,Z 354.204,A -85,B 0,C 180,E1 27359.592,E2 27359.592} C_VEL
LIN {X 0,Y 568.139,Z 354.209,A -85,B 0,C 180,E1 27356.464,E2 27356.464} C_VEL
LIN {X 0,Y 568.211,Z 354.2,A -85,B 0,C 180,E1 27353.327,E2 27353.327} C_VEL
LIN {X 0,Y 568.141,Z 354.209,A -85,B 0,C 180,E1 27350.231,E2 27350.231} C_VEL
LIN {X 0,Y 568.177,Z 354.201,A -85,B 0,C 180,E1 27346.979,E2 27346.979} C_VEL
LIN {X 0,Y 568.144,Z 354.206,A -85,B 0,C 180,E1 27344.062,E2 27344.062} C_VEL
LIN {X 0,Y 568.167,Z 354.206,A -85,B 0,C 180,E1 27340.784,E2 27340.784} C_VEL
LIN {X 0,Y 568.148,Z 354.202,A -85,B 0,C 180,E1 27337.873,E2 27337.873} C_VEL
LIN {X 0,Y 568.15,Z 354.208,A -85,B 0,C 180,E1 27334.456,E2 27334.456} C_VEL
LIN {X 0,Y 568.168,Z 354.201,A -85,B 0,C 180,E1 27331.514,E2 27331.514} C_VEL
LIN {X 0,Y 568.146,Z 354.208,A -85,B 0,C 180,E1 27328.248,E2 27328.248} C_VEL
LIN {X 0,Y 568.212,Z 354.207,A -85,B 0,C 180,E1 27325.082,E2 27325.082} C_VEL
LIN {X 0,Y 568.141,Z 354.206,A -85,B 0,C 180,E1 27321.976,E2 27321.976} C_VEL
LIN {X 0,Y 568.219,Z 354.205,A -85,B 0,C 180,E1 27318.842,E2 27318.842} C_VEL
LIN {X 0,Y 568.145,Z 354.209,A -85,B 0,C 180,E1 27315.678,E2 27315.678} C_VEL
LIN {X 0,Y 568.188,Z 354.203,A -85,B 0,C 180,E1 27312.494,E2 27312.494} C_VEL
LIN {X 0,Y 568.145,Z 354.208,A -85,B 0,C 180,E1 27309.57,E2 27309.57} C_VEL
LIN {X 0,Y 568.176,Z 354.193,A -85,B 0,C 180,E1 27306.294,E2 27306.294} C_VEL
LIN {X 0,Y 568.247,Z 354.504,A -85,B 0,C 180,E1 27304.784,E2 27304.784} C_VEL
LIN {X 0,Y 570.848,Z 364.504,A -85,B 0,C 180,E1 27303.333,E2 27303.333} C_VEL
LIN {X 0,Y 570.33,Z 390.222,A -85,B 0,C 180,E1 27300.197,E2 27300.197} C_VEL
LIN {X 0,Y 570.349,Z 395.301,A -85,B 0,C 180,E1 27299.631,E2 27299.631} C_VEL
LIN {X 0,Y 572.636,Z 404.319,A -85,B 0,C 180,E1 27299.369,E2 27299.369} C_VEL
LIN {X 0,Y 571.7,Z 639.159,A -85,B 0,C 180,E1 27296.155,E2 27296.155} C_VEL
LIN {X 0,Y 571.518,Z 661.766,A -85,B 0,C 180,E1 27295.765,E2 27295.765} C_VEL
LIN {X 0,Y 571.217,Z 682.048,A -85,B 0,C 180,E1 27295.226,E2 27295.226} C_VEL
LIN {X 0,Y 570.862,Z 702.738,A -85,B 0,C 180,E1 27294.47,E2 27294.47} C_VEL
LIN {X 0,Y 570.508,Z 721.262,A -85,B 0,C 180,E1 27293.606,E2 27293.606} C_VEL
LIN {X 0,Y 570.106,Z 740.269,A -85,B 0,C 180,E1 27292.52,E2 27292.52} C_VEL
LIN {X 0,Y 569.67,Z 757.797,A -85,B 0,C 180,E1 27291.303,E2 27291.303} C_VEL
LIN {X 0,Y 569.278,Z 774.665,A -85,B 0,C 180,E1 27289.921,E2 27289.921} C_VEL
LIN {X 0,Y 568.917,Z 790.647,A -85,B 0,C 180,E1 27288.369,E2 27288.369} C_VEL
LIN {X 0,Y 568.621,Z 804.775,A -85,B 0,C 180,E1 27286.76,E2 27286.76} C_VEL
LIN {X 0,Y 568.371,Z 817.975,A -85,B 0,C 180,E1 27284.986,E2 27284.986} C_VEL
LIN {X 0,Y 568.207,Z 829.121,A -85,B 0,C 180,E1 27283.224,E2 27283.224} C_VEL
LIN {X 0,Y 568.068,Z 839.391,A -85,B 0,C 180,E1 27281.266,E2 27281.266} C_VEL
LIN {X 0,Y 567.992,Z 847.678,A -85,B 0,C 180,E1 27279.32,E2 27279.32} C_VEL
LIN {X 0,Y 567.942,Z 854.524,A -85,B 0,C 180,E1 27277.282,E2 27277.282} C_VEL
LIN {X 0,Y 567.917,Z 859.543,A -85,B 0,C 180,E1 27275.253,E2 27275.253} C_VEL
LIN {X 0,Y 567.911,Z 862.96,A -85,B 0,C 180,E1 27273.23,E2 27273.23} C_VEL
LIN {X 0,Y 567.911,Z 864.741,A -85,B 0,C 180,E1 27271.11,E2 27271.11} C_VEL
LIN {X 0,Y 567.914,Z 864.799,A -85,B 0,C 180,E1 27269.092,E2 27269.092} C_VEL
LIN {X 0,Y 567.915,Z 863.296,A -85,B 0,C 180,E1 27267.073,E2 27267.073} C_VEL
LIN {X 0,Y 567.922,Z 859.953,A -85,B 0,C 180,E1 27264.95,E2 27264.95} C_VEL
LIN {X 0,Y 567.943,Z 855.13,A -85,B 0,C 180,E1 27262.921,E2 27262.921} C_VEL
LIN {X 0,Y 567.982,Z 848.469,A -85,B 0,C 180,E1 27260.884,E2 27260.884} C_VEL
LIN {X 0,Y 568.048,Z 840.32,A -85,B 0,C 180,E1 27258.939,E2 27258.939} C_VEL
LIN {X 0,Y 568.181,Z 830.281,A -85,B 0,C 180,E1 27256.983,E2 27256.983} C_VEL
LIN {X 0,Y 568.36,Z 818.681,A -85,B 0,C 180,E1 27255.118,E2 27255.118} C_VEL
LIN {X 0,Y 568.601,Z 805.624,A -85,B 0,C 180,E1 27253.344,E2 27253.344} C_VEL
LIN {X 0,Y 568.91,Z 790.964,A -85,B 0,C 180,E1 27251.664,E2 27251.664} C_VEL
LIN {X 0,Y 569.261,Z 775.496,A -85,B 0,C 180,E1 27250.152,E2 27250.152} C_VEL
LIN {X 0,Y 569.658,Z 758.518,A -85,B 0,C 180,E1 27248.751,E2 27248.751} C_VEL
LIN {X 0,Y 570.088,Z 740.9,A -85,B 0,C 180,E1 27247.522,E2 27247.522} C_VEL
LIN {X 0,Y 570.49,Z 722.155,A -85,B 0,C 180,E1 27246.439,E2 27246.439} C_VEL
LIN {X 0,Y 570.832,Z 704.012,A -85,B 0,C 180,E1 27245.584,E2 27245.584} C_VEL
LIN {X 0,Y 571.213,Z 682.474,A -85,B 0,C 180,E1 27244.788,E2 27244.788} C_VEL
LIN {X 0,Y 571.507,Z 662.503,A -85,B 0,C 180,E1 27244.252,E2 27244.252} C_VEL
LIN {X 0,Y 571.693,Z 641.101,A -85,B 0,C 180,E1 27243.871,E2 27243.871} C_VEL
LIN {X 0,Y 572.629,Z 406.228,A -85,B 0,C 180,E1 27240.657,E2 27240.657} C_VEL
LIN {X 0,Y 572.378,Z 402.613,A -85,B 0,C 180,E1 27240.592,E2 27240.592} C_VEL
LIN {X 0,Y 570.266,Z 394.633,A -85,B 0,C 180,E1 27240.325,E2 27240.325} C_VEL
LIN {X 0,Y 570.775,Z 368.084,A -85,B 0,C 180,E1 27237.11,E2 27237.11} C_VEL
LIN {X 0,Y 570.737,Z 363.244,A -85,B 0,C 180,E1 27236.502,E2 27236.502} C_VEL
LIN {X 0,Y 568.207,Z 354.282,A -85,B 0,C 180,E1 27235.15,E2 27235.15} C_VEL
LIN {X 0,Y 568.146,Z 354.208,A -85,B 0,C 180,E1 27232.108,E2 27232.108} C_VEL
LIN {X 0,Y 568.172,Z 354.2,A -85,B 0,C 180,E1 27228.842,E2 27228.842} C_VEL
LIN {X 0,Y 568.155,Z 354.21,A -85,B 0,C 180,E1 27225.823,E2 27225.823} C_VEL
LIN {X 0,Y 568.152,Z 354.208,A -85,B 0,C 180,E1 27222.494,E2 27222.494} C_VEL
LIN {X 0,Y 568.168,Z 354.209,A -85,B 0,C 180,E1 27219.574,E2 27219.574} C_VEL
LIN {X 0,Y 568.147,Z 354.21,A -85,B 0,C 180,E1 27216.294,E2 27216.294} C_VEL
LIN {X 0,Y 568.186,Z 354.206,A -85,B 0,C 180,E1 27213.296,E2 27213.296} C_VEL
LIN {X 0,Y 568.144,Z 354.209,A -85,B 0,C 180,E1 27210.106,E2 27210.106} C_VEL
LIN {X 0,Y 568.208,Z 354.2,A -85,B 0,C 180,E1 27207.003,E2 27207.003} C_VEL
LIN {X 0,Y 568.141,Z 354.209,A -85,B 0,C 180,E1 27203.88,E2 27203.88} C_VEL
LIN {X 0,Y 568.211,Z 354.202,A -85,B 0,C 180,E1 27200.716,E2 27200.716} C_VEL
LIN {X 0,Y 568.141,Z 354.209,A -85,B 0,C 180,E1 27197.623,E2 27197.623} C_VEL
LIN {X 0,Y 568.192,Z 354.201,A -85,B 0,C 180,E1 27194.474,E2 27194.474} C_VEL
LIN {X 0,Y 568.145,Z 354.208,A -85,B 0,C 180,E1 27191.416,E2 27191.416} C_VEL
LIN {X 0,Y 568.161,Z 354.204,A -85,B 0,C 180,E1 27188.097,E2 27188.097} C_VEL
LIN {X 0,Y 568.156,Z 354.202,A -85,B 0,C 180,E1 27185.104,E2 27185.104} C_VEL
LIN {X 0,Y 568.148,Z 354.209,A -85,B 0,C 180,E1 27181.82,E2 27181.82} C_VEL
LIN {X 0,Y 568.163,Z 354.203,A -85,B 0,C 180,E1 27178.895,E2 27178.895} C_VEL
LIN {X 0,Y 568.146,Z 354.209,A -85,B 0,C 180,E1 27175.665,E2 27175.665} C_VEL
LIN {X 0,Y 568.183,Z 354.208,A -85,B 0,C 180,E1 27172.624,E2 27172.624} C_VEL
LIN {X 0,Y 568.14,Z 354.205,A -85,B 0,C 180,E1 27169.459,E2 27169.459} C_VEL
LIN {X 0,Y 568.205,Z 354.209,A -85,B 0,C 180,E1 27166.367,E2 27166.367} C_VEL
LIN {X 0,Y 568.137,Z 354.2,A -85,B 0,C 180,E1 27163.206,E2 27163.206} C_VEL
LIN {X 0,Y 568.207,Z 354.211,A -85,B 0,C 180,E1 27160.045,E2 27160.045} C_VEL
LIN {X 0,Y 568.182,Z 354.21,A -85,B 0,C 180,E1 27159.834,E2 27159.834} C_VEL
LIN {X 0,Y 567.127,Z 354.337,A -85,B 0,C 180,E1 27159.058,E2 27159.058} C_VEL
LIN {X 0,Y 560.724,Z 355.137,A -85,B 0,C 180,E1 27156.878,E2 27156.878} C_VEL
LIN {X 0,Y 560.249,Z 355.192,A -85,B 0,C 180,E1 27156.31,E2 27156.31} C_VEL
LIN {X 0,Y 560.199,Z 355.199,A -85,B 0,C 180,E1 27153.163,E2 27153.163} C_VEL
LIN {X 0,Y 560.278,Z 355.198,A -85,B 0,C 180,E1 27150.029,E2 27150.029} C_VEL
LIN {X 0,Y 560.199,Z 355.199,A -85,B 0,C 180,E1 27146.831,E2 27146.831} C_VEL
LIN {X 0,Y 560.244,Z 355.199,A -85,B 0,C 180,E1 27143.598,E2 27143.598} C_VEL
LIN {X 0,Y 560.203,Z 355.199,A -85,B 0,C 180,E1 27140.56,E2 27140.56} C_VEL
LIN {X 0,Y 560.211,Z 355.2,A -85,B 0,C 180,E1 27137.166,E2 27137.166} C_VEL
LIN {X 0,Y 560.23,Z 355.199,A -85,B 0,C 180,E1 27134.109,E2 27134.109} C_VEL
LIN {X 0,Y 560.199,Z 355.199,A -85,B 0,C 180,E1 27130.832,E2 27130.832} C_VEL
LIN {X 0,Y 560.263,Z 355.199,A -85,B 0,C 180,E1 27127.742,E2 27127.742} C_VEL
LIN {X 0,Y 560.197,Z 355.2,A -85,B 0,C 180,E1 27124.58,E2 27124.58} C_VEL
LIN {X 0,Y 560.265,Z 355.2,A -85,B 0,C 180,E1 27121.406,E2 27121.406} C_VEL
LIN {X 0,Y 560.198,Z 355.199,A -85,B 0,C 180,E1 27118.343,E2 27118.343} C_VEL
LIN {X 0,Y 560.243,Z 355.2,A -85,B 0,C 180,E1 27115.134,E2 27115.134} C_VEL
LIN {X 0,Y 560.201,Z 355.199,A -85,B 0,C 180,E1 27112.122,E2 27112.122} C_VEL
LIN {X 0,Y 560.211,Z 355.2,A -85,B 0,C 180,E1 27108.739,E2 27108.739} C_VEL
LIN {X 0,Y 560.218,Z 355.2,A -85,B 0,C 180,E1 27105.74,E2 27105.74} C_VEL
LIN {X 0,Y 560.202,Z 355.199,A -85,B 0,C 180,E1 27102.472,E2 27102.472} C_VEL
LIN {X 0,Y 560.253,Z 355.2,A -85,B 0,C 180,E1 27099.332,E2 27099.332} C_VEL
LIN {X 0,Y 560.194,Z 355.2,A -85,B 0,C 180,E1 27096.147,E2 27096.147} C_VEL
LIN {X 0,Y 560.261,Z 355.199,A -85,B 0,C 180,E1 27092.967,E2 27092.967} C_VEL
LIN {X 0,Y 560.194,Z 355.2,A -85,B 0,C 180,E1 27089.898,E2 27089.898} C_VEL
LIN {X 0,Y 560.246,Z 355.199,A -85,B 0,C 180,E1 27086.726,E2 27086.726} C_VEL
LIN {X 0,Y 560.2,Z 355.2,A -85,B 0,C 180,E1 27083.647,E2 27083.647} C_VEL
LIN {X 0,Y 560.217,Z 355.2,A -85,B 0,C 180,E1 27080.342,E2 27080.342} C_VEL
LIN {X 0,Y 560.214,Z 355.199,A -85,B 0,C 180,E1 27077.319,E2 27077.319} C_VEL
LIN {X 0,Y 560.203,Z 355.2,A -85,B 0,C 180,E1 27074.047,E2 27074.047} C_VEL
LIN {X 0,Y 560.244,Z 355.2,A -85,B 0,C 180,E1 27070.938,E2 27070.938} C_VEL
LIN {X 0,Y 560.198,Z 355.2,A -85,B 0,C 180,E1 27067.767,E2 27067.767} C_VEL
LIN {X 0,Y 560.266,Z 355.199,A -85,B 0,C 180,E1 27064.641,E2 27064.641} C_VEL
LIN {X 0,Y 560.196,Z 355.199,A -85,B 0,C 180,E1 27061.541,E2 27061.541} C_VEL
LIN {X 0,Y 560.258,Z 355.199,A -85,B 0,C 180,E1 27058.335,E2 27058.335} C_VEL
LIN {X 0,Y 560.198,Z 355.2,A -85,B 0,C 180,E1 27055.296,E2 27055.296} C_VEL
LIN {X 0,Y 560.237,Z 355.199,A -85,B 0,C 180,E1 27052.065,E2 27052.065} C_VEL
LIN {X 0,Y 560.205,Z 355.199,A -85,B 0,C 180,E1 27049.011,E2 27049.011} C_VEL
LIN {X 0,Y 560.207,Z 355.199,A -85,B 0,C 180,E1 27045.603,E2 27045.603} C_VEL
LIN {X 0,Y 560.241,Z 355.2,A -85,B 0,C 180,E1 27042.519,E2 27042.519} C_VEL
LIN {X 0,Y 560.198,Z 355.199,A -85,B 0,C 180,E1 27039.308,E2 27039.308} C_VEL
LIN {X 0,Y 560.269,Z 355.199,A -85,B 0,C 180,E1 27036.198,E2 27036.198} C_VEL
LIN {X 0,Y 560.199,Z 355.199,A -85,B 0,C 180,E1 27033.096,E2 27033.096} C_VEL
LIN {X 0,Y 560.278,Z 355.198,A -85,B 0,C 180,E1 27029.971,E2 27029.971} C_VEL
LIN {X 0,Y 560.2,Z 355.199,A -85,B 0,C 180,E1 27026.826,E2 27026.826} C_VEL
LIN {X 0,Y 560.235,Z 355.193,A -85,B 0,C 180,E1 27023.557,E2 27023.557} C_VEL
LIN {X 0,Y 560.207,Z 355.199,A -85,B 0,C 180,E1 27020.579,E2 27020.579} C_VEL
LIN {X 0,Y 560.206,Z 355.188,A -85,B 0,C 180,E1 27017.121,E2 27017.121} C_VEL
LIN {X 0,Y 560.232,Z 355.197,A -85,B 0,C 180,E1 27014.147,E2 27014.147} C_VEL
LIN {X 0,Y 560.202,Z 355.193,A -85,B 0,C 180,E1 27010.9,E2 27010.9} C_VEL
LIN {X 0,Y 560.28,Z 355.191,A -85,B 0,C 180,E1 27007.687,E2 27007.687} C_VEL
LIN {X 0,Y 560.202,Z 355.198,A -85,B 0,C 180,E1 27004.499,E2 27004.499} C_VEL
LIN {X 0,Y 560.236,Z 355.19,A -85,B 0,C 180,E1 27001.223,E2 27001.223} C_VEL
LIN {X 0,Y 560.206,Z 355.198,A -85,B 0,C 180,E1 26998.257,E2 26998.257} C_VEL
LIN {X 0,Y 560.216,Z 355.19,A -85,B 0,C 180,E1 26994.876,E2 26994.876} C_VEL
LIN {X 0,Y 560.223,Z 355.192,A -85,B 0,C 180,E1 26991.891,E2 26991.891} C_VEL
LIN {X 0,Y 560.206,Z 355.197,A -85,B 0,C 180,E1 26988.57,E2 26988.57} C_VEL
LIN {X 0,Y 560.267,Z 355.187,A -85,B 0,C 180,E1 26985.423,E2 26985.423} C_VEL
LIN {X 0,Y 560.2,Z 355.199,A -85,B 0,C 180,E1 26982.226,E2 26982.226} C_VEL
LIN {X 0,Y 560.269,Z 355.187,A -85,B 0,C 180,E1 26979.086,E2 26979.086} C_VEL
LIN {X 0,Y 560.204,Z 355.198,A -85,B 0,C 180,E1 26975.984,E2 26975.984} C_VEL
LIN {X 0,Y 560.233,Z 355.188,A -85,B 0,C 180,E1 26972.696,E2 26972.696} C_VEL
LIN {X 0,Y 560.216,Z 355.198,A -85,B 0,C 180,E1 26969.66,E2 26969.66} C_VEL
LIN {X 0,Y 560.209,Z 355.195,A -85,B 0,C 180,E1 26966.273,E2 26966.273} C_VEL
LIN {X 0,Y 560.245,Z 355.199,A -85,B 0,C 180,E1 26963.254,E2 26963.254} C_VEL
LIN {X 0,Y 560.205,Z 355.199,A -85,B 0,C 180,E1 26960.017,E2 26960.017} C_VEL
LIN {X 0,Y 560.278,Z 355.199,A -85,B 0,C 180,E1 26956.875,E2 26956.875} C_VEL
LIN {X 0,Y 560.205,Z 355.2,A -85,B 0,C 180,E1 26953.686,E2 26953.686} C_VEL
LIN {X 0,Y 560.255,Z 355.183,A -85,B 0,C 180,E1 26950.511,E2 26950.511} C_VEL
LIN {X 0,Y 560.208,Z 355.195,A -85,B 0,C 180,E1 26947.488,E2 26947.488} C_VEL
LIN {X 0,Y 560.239,Z 355.341,A -85,B 0,C 180,E1 26945.232,E2 26945.232} C_VEL
LIN {X 0,Y 563.443,Z 367.227,A -85,B 0,C 180,E1 26943.482,E2 26943.482} C_VEL
LIN {X 0,Y 562.805,Z 393.491,A -85,B 0,C 180,E1 26940.241,E2 26940.241} C_VEL
LIN {X 0,Y 562.936,Z 395.599,A -85,B 0,C 180,E1 26940.053,E2 26940.053} C_VEL
LIN {X 0,Y 565.655,Z 406.026,A -85,B 0,C 180,E1 26939.744,E2 26939.744} C_VEL
LIN {X 0,Y 564.511,Z 640.974,A -85,B 0,C 180,E1 26936.489,E2 26936.489} C_VEL
LIN {X 0,Y 564.286,Z 662.32,A -85,B 0,C 180,E1 26936.106,E2 26936.106} C_VEL
LIN {X 0,Y 563.942,Z 682.126,A -85,B 0,C 180,E1 26935.572,E2 26935.572} C_VEL
LIN {X 0,Y 563.523,Z 702.741,A -85,B 0,C 180,E1 26934.81,E2 26934.81} C_VEL
LIN {X 0,Y 563.108,Z 720.184,A -85,B 0,C 180,E1 26933.992,E2 26933.992} C_VEL
LIN {X 0,Y 562.632,Z 738.24,A -85,B 0,C 180,E1 26932.964,E2 26932.964} C_VEL
LIN {X 0,Y 562.119,Z 756.37,A -85,B 0,C 180,E1 26931.713,E2 26931.713} C_VEL
LIN {X 0,Y 561.639,Z 773.464,A -85,B 0,C 180,E1 26930.312,E2 26930.312} C_VEL
LIN {X 0,Y 561.174,Z 789.961,A -85,B 0,C 180,E1 26928.705,E2 26928.705} C_VEL
LIN {X 0,Y 560.795,Z 804.779,A -85,B 0,C 180,E1 26927.001,E2 26927.001} C_VEL
LIN {X 0,Y 560.478,Z 818.14,A -85,B 0,C 180,E1 26925.178,E2 26925.178} C_VEL
LIN {X 0,Y 560.265,Z 829.708,A -85,B 0,C 180,E1 26923.309,E2 26923.309} C_VEL
LIN {X 0,Y 560.097,Z 839.852,A -85,B 0,C 180,E1 26921.324,E2 26921.324} C_VEL
LIN {X 0,Y 560.007,Z 847.674,A -85,B 0,C 180,E1 26919.454,E2 26919.454} C_VEL
LIN {X 0,Y 559.948,Z 854.528,A -85,B 0,C 180,E1 26917.386,E2 26917.386} C_VEL
LIN {X 0,Y 559.918,Z 859.541,A -85,B 0,C 180,E1 26915.328,E2 26915.328} C_VEL
LIN {X 0,Y 559.91,Z 862.963,A -85,B 0,C 180,E1 26913.276,E2 26913.276} C_VEL
LIN {X 0,Y 559.911,Z 864.737,A -85,B 0,C 180,E1 26911.126,E2 26911.126} C_VEL
LIN {X 0,Y 559.914,Z 864.795,A -85,B 0,C 180,E1 26909.079,E2 26909.079} C_VEL
LIN {X 0,Y 559.915,Z 863.187,A -85,B 0,C 180,E1 26906.929,E2 26906.929} C_VEL
LIN {X 0,Y 559.922,Z 859.951,A -85,B 0,C 180,E1 26904.878,E2 26904.878} C_VEL
LIN {X 0,Y 559.949,Z 855.133,A -85,B 0,C 180,E1 26902.82,E2 26902.82} C_VEL
LIN {X 0,Y 560.006,Z 848.069,A -85,B 0,C 180,E1 26900.65,E2 26900.65} C_VEL
LIN {X 0,Y 560.087,Z 840.317,A -85,B 0,C 180,E1 26898.78,E2 26898.78} C_VEL
LIN {X 0,Y 560.251,Z 830.285,A -85,B 0,C 180,E1 26896.795,E2 26896.795} C_VEL
LIN {X 0,Y 560.467,Z 818.681,A -85,B 0,C 180,E1 26894.903,E2 26894.903} C_VEL
LIN {X 0,Y 560.77,Z 805.628,A -85,B 0,C 180,E1 26893.105,E2 26893.105} C_VEL
LIN {X 0,Y 561.136,Z 791.249,A -85,B 0,C 180,E1 26891.433,E2 26891.433} C_VEL
LIN {X 0,Y 561.565,Z 775.877,A -85,B 0,C 180,E1 26889.902,E2 26889.902} C_VEL
LIN {X 0,Y 562.047,Z 758.566,A -85,B 0,C 180,E1 26888.454,E2 26888.454} C_VEL
LIN {X 0,Y 562.543,Z 741.699,A -85,B 0,C 180,E1 26887.259,E2 26887.259} C_VEL
LIN {X 0,Y 563.06,Z 722.304,A -85,B 0,C 180,E1 26886.118,E2 26886.118} C_VEL
LIN {X 0,Y 563.485,Z 704.011,A -85,B 0,C 180,E1 26885.244,E2 26885.244} C_VEL
LIN {X 0,Y 563.938,Z 682.368,A -85,B 0,C 180,E1 26884.436,E2 26884.436} C_VEL
LIN {X 0,Y 564.282,Z 662.614,A -85,B 0,C 180,E1 26883.901,E2 26883.901} C_VEL
LIN {X 0,Y 564.51,Z 641.355,A -85,B 0,C 180,E1 26883.516,E2 26883.516} C_VEL
LIN {X 0,Y 565.654,Z 406.423,A -85,B 0,C 180,E1 26880.262,E2 26880.262} C_VEL
LIN {X 0,Y 564.894,Z 402.494,A -85,B 0,C 180,E1 26880.162,E2 26880.162} C_VEL
LIN {X 0,Y 562.806,Z 394.808,A -85,B 0,C 180,E1 26879.905,E2 26879.905} C_VEL
LIN {X 0,Y 563.404,Z 368.749,A -85,B 0,C 180,E1 26876.708,E2 26876.708} C_VEL
LIN {X 0,Y 563.161,Z 365.55,A -85,B 0,C 180,E1 26876.285,E2 26876.285} C_VEL
LIN {X 0,Y 560.226,Z 355.263,A -85,B 0,C 180,E1 26874.736,E2 26874.736} C_VEL
LIN {X 0,Y 560.233,Z 355.197,A -85,B 0,C 180,E1 26871.737,E2 26871.737} C_VEL
LIN {X 0,Y 560.21,Z 355.191,A -85,B 0,C 180,E1 26868.537,E2 26868.537} C_VEL
LIN {X 0,Y 560.259,Z 355.199,A -85,B 0,C 180,E1 26865.406,E2 26865.406} C_VEL
LIN {X 0,Y 560.204,Z 355.197,A -85,B 0,C 180,E1 26862.211,E2 26862.211} C_VEL
LIN {X 0,Y 560.281,Z 355.196,A -85,B 0,C 180,E1 26859.049,E2 26859.049} C_VEL
LIN {X 0,Y 560.205,Z 355.198,A -85,B 0,C 180,E1 26855.877,E2 26855.877} C_VEL
LIN {X 0,Y 560.236,Z 355.198,A -85,B 0,C 180,E1 26852.61,E2 26852.61} C_VEL
LIN {X 0,Y 560.212,Z 355.197,A -85,B 0,C 180,E1 26849.632,E2 26849.632} C_VEL
LIN {X 0,Y 560.215,Z 355.198,A -85,B 0,C 180,E1 26846.274,E2 26846.274} C_VEL
LIN {X 0,Y 560.237,Z 355.197,A -85,B 0,C 180,E1 26843.206,E2 26843.206} C_VEL
LIN {X 0,Y 560.203,Z 355.195,A -85,B 0,C 180,E1 26839.935,E2 26839.935} C_VEL
LIN {X 0,Y 560.274,Z 355.198,A -85,B 0,C 180,E1 26836.808,E2 26836.808} C_VEL
LIN {X 0,Y 560.201,Z 355.189,A -85,B 0,C 180,E1 26833.63,E2 26833.63} C_VEL
LIN {X 0,Y 560.251,Z 355.199,A -85,B 0,C 180,E1 26830.388,E2 26830.388} C_VEL
LIN {X 0,Y 560.208,Z 355.191,A -85,B 0,C 180,E1 26827.284,E2 26827.284} C_VEL
LIN {X 0,Y 560.213,Z 355.198,A -85,B 0,C 180,E1 26823.893,E2 26823.893} C_VEL
LIN {X 0,Y 560.239,Z 355.197,A -85,B 0,C 180,E1 26820.822,E2 26820.822} C_VEL
LIN {X 0,Y 560.2,Z 355.191,A -85,B 0,C 180,E1 26817.55,E2 26817.55} C_VEL
LIN {X 0,Y 560.275,Z 355.198,A -85,B 0,C 180,E1 26814.372,E2 26814.372} C_VEL
LIN {X 0,Y 560.199,Z 355.19,A -85,B 0,C 180,E1 26811.279,E2 26811.279} C_VEL
LIN {X 0,Y 560.254,Z 355.199,A -85,B 0,C 180,E1 26808.058,E2 26808.058} C_VEL
LIN {X 0,Y 560.201,Z 355.197,A -85,B 0,C 180,E1 26805.007,E2 26805.007} C_VEL
LIN {X 0,Y 560.224,Z 355.196,A -85,B 0,C 180,E1 26801.699,E2 26801.699} C_VEL
LIN {X 0,Y 560.218,Z 355.198,A -85,B 0,C 180,E1 26798.655,E2 26798.655} C_VEL
LIN {X 0,Y 560.249,Z 355.192,A -85,B 0,C 180,E1 26796.31,E2 26796.31} C_VEL
LIN {X 0,Y 559.306,Z 355.307,A -85,B 0,C 180,E1 26795.522,E2 26795.522} C_VEL
LIN {X 0,Y 552.792,Z 356.125,A -85,B 0,C 180,E1 26793.311,E2 26793.311} C_VEL
LIN {X 0,Y 552.267,Z 356.188,A -85,B 0,C 180,E1 26792.734,E2 26792.734} C_VEL
LIN {X 0,Y 552.271,Z 356.188,A -85,B 0,C 180,E1 26789.307,E2 26789.307} C_VEL
LIN {X 0,Y 552.299,Z 356.188,A -85,B 0,C 180,E1 26786.244,E2 26786.244} C_VEL
LIN {X 0,Y 552.26,Z 356.187,A -85,B 0,C 180,E1 26782.978,E2 26782.978} C_VEL
LIN {X 0,Y 552.331,Z 356.188,A -85,B 0,C 180,E1 26779.81,E2 26779.81} C_VEL
LIN {X 0,Y 552.259,Z 356.188,A -85,B 0,C 180,E1 26776.682,E2 26776.682} C_VEL
LIN {X 0,Y 552.308,Z 356.189,A -85,B 0,C 180,E1 26773.464,E2 26773.464} C_VEL
LIN {X 0,Y 552.266,Z 356.188,A -85,B 0,C 180,E1 26770.353,E2 26770.353} C_VEL
LIN {X 0,Y 552.268,Z 356.189,A -85,B 0,C 180,E1 26766.945,E2 26766.945} C_VEL
LIN {X 0,Y 552.312,Z 356.189,A -85,B 0,C 180,E1 26763.762,E2 26763.762} C_VEL
LIN {X 0,Y 552.257,Z 356.188,A -85,B 0,C 180,E1 26760.579,E2 26760.579} C_VEL
LIN {X 0,Y 552.328,Z 356.188,A -85,B 0,C 180,E1 26757.374,E2 26757.374} C_VEL
LIN {X 0,Y 552.262,Z 356.189,A -85,B 0,C 180,E1 26754.152,E2 26754.152} C_VEL
LIN {X 0,Y 552.274,Z 356.188,A -85,B 0,C 180,E1 26750.783,E2 26750.783} C_VEL
LIN {X 0,Y 552.287,Z 356.189,A -85,B 0,C 180,E1 26747.706,E2 26747.706} C_VEL
LIN {X 0,Y 552.259,Z 356.189,A -85,B 0,C 180,E1 26744.428,E2 26744.428} C_VEL
LIN {X 0,Y 552.322,Z 356.189,A -85,B 0,C 180,E1 26741.274,E2 26741.274} C_VEL
LIN {X 0,Y 552.255,Z 356.19,A -85,B 0,C 180,E1 26738.118,E2 26738.118} C_VEL
LIN {X 0,Y 552.323,Z 356.189,A -85,B 0,C 180,E1 26734.985,E2 26734.985} C_VEL
LIN {X 0,Y 552.261,Z 356.189,A -85,B 0,C 180,E1 26731.764,E2 26731.764} C_VEL
LIN {X 0,Y 552.267,Z 356.189,A -85,B 0,C 180,E1 26728.34,E2 26728.34} C_VEL
LIN {X 0,Y 552.298,Z 356.188,A -85,B 0,C 180,E1 26725.223,E2 26725.223} C_VEL
LIN {X 0,Y 552.257,Z 356.189,A -85,B 0,C 180,E1 26721.987,E2 26721.987} C_VEL
LIN {X 0,Y 552.326,Z 356.189,A -85,B 0,C 180,E1 26718.818,E2 26718.818} C_VEL
LIN {X 0,Y 552.257,Z 356.189,A -85,B 0,C 180,E1 26715.639,E2 26715.639} C_VEL
LIN {X 0,Y 552.298,Z 356.189,A -85,B 0,C 180,E1 26712.403,E2 26712.403} C_VEL
LIN {X 0,Y 552.266,Z 356.188,A -85,B 0,C 180,E1 26709.327,E2 26709.327} C_VEL
LIN {X 0,Y 552.267,Z 356.189,A -85,B 0,C 180,E1 26705.962,E2 26705.962} C_VEL
LIN {X 0,Y 552.3,Z 356.189,A -85,B 0,C 180,E1 26702.858,E2 26702.858} C_VEL
LIN {X 0,Y 552.259,Z 356.188,A -85,B 0,C 180,E1 26699.661,E2 26699.661} C_VEL
LIN {X 0,Y 552.33,Z 356.188,A -85,B 0,C 180,E1 26696.488,E2 26696.488} C_VEL
LIN {X 0,Y 552.258,Z 356.189,A -85,B 0,C 180,E1 26693.313,E2 26693.313} C_VEL
LIN {X 0,Y 552.31,Z 356.188,A -85,B 0,C 180,E1 26690.125,E2 26690.125} C_VEL
LIN {X 0,Y 552.262,Z 356.188,A -85,B 0,C 180,E1 26687.1,E2 26687.1} C_VEL
LIN {X 0,Y 552.28,Z 356.188,A -85,B 0,C 180,E1 26683.745,E2 26683.745} C_VEL
LIN {X 0,Y 552.273,Z 356.188,A -85,B 0,C 180,E1 26680.802,E2 26680.802} C_VEL
LIN {X 0,Y 552.267,Z 356.187,A -85,B 0,C 180,E1 26677.459,E2 26677.459} C_VEL
LIN {X 0,Y 552.305,Z 356.189,A -85,B 0,C 180,E1 26674.362,E2 26674.362} C_VEL
LIN {X 0,Y 552.261,Z 356.188,A -85,B 0,C 180,E1 26671.177,E2 26671.177} C_VEL
LIN {X 0,Y 552.33,Z 356.189,A -85,B 0,C 180,E1 26668.07,E2 26668.07} C_VEL
LIN {X 0,Y 552.26,Z 356.182,A -85,B 0,C 180,E1 26664.83,E2 26664.83} C_VEL
LIN {X 0,Y 552.299,Z 356.187,A -85,B 0,C 180,E1 26661.555,E2 26661.555} C_VEL
LIN {X 0,Y 552.275,Z 356.185,A -85,B 0,C 180,E1 26658.443,E2 26658.443} C_VEL
LIN {X 0,Y 552.268,Z 356.185,A -85,B 0,C 180,E1 26655.106,E2 26655.106} C_VEL
LIN {X 0,Y 552.306,Z 356.188,A -85,B 0,C 180,E1 26652.011,E2 26652.011} C_VEL
LIN {X 0,Y 552.261,Z 356.177,A -85,B 0,C 180,E1 26648.742,E2 26648.742} C_VEL
LIN {X 0,Y 552.334,Z 356.187,A -85,B 0,C 180,E1 26645.605,E2 26645.605} C_VEL
LIN {X 0,Y 552.263,Z 356.179,A -85,B 0,C 180,E1 26642.382,E2 26642.382} C_VEL
LIN {X 0,Y 552.287,Z 356.186,A -85,B 0,C 180,E1 26639.062,E2 26639.062} C_VEL
LIN {X 0,Y 552.286,Z 356.187,A -85,B 0,C 180,E1 26635.947,E2 26635.947} C_VEL
LIN {X 0,Y 552.265,Z 356.18,A -85,B 0,C 180,E1 26632.611,E2 26632.611} C_VEL
LIN {X 0,Y 552.333,Z 356.188,A -85,B 0,C 180,E1 26629.399,E2 26629.399} C_VEL
LIN {X 0,Y 552.263,Z 356.177,A -85,B 0,C 180,E1 26626.17,E2 26626.17} C_VEL
LIN {X 0,Y 552.298,Z 356.187,A -85,B 0,C 180,E1 26622.909,E2 26622.909} C_VEL
LIN {X 0,Y 552.273,Z 356.184,A -85,B 0,C 180,E1 26619.877,E2 26619.877} C_VEL
LIN {X 0,Y 552.275,Z 356.186,A -85,B 0,C 180,E1 26616.525,E2 26616.525} C_VEL
LIN {X 0,Y 552.305,Z 356.187,A -85,B 0,C 180,E1 26613.416,E2 26613.416} C_VEL
LIN {X 0,Y 552.268,Z 356.186,A -85,B 0,C 180,E1 26610.257,E2 26610.257} C_VEL
LIN {X 0,Y 552.329,Z 356.182,A -85,B 0,C 180,E1 26607.104,E2 26607.104} C_VEL
LIN {X 0,Y 552.265,Z 356.188,A -85,B 0,C 180,E1 26603.954,E2 26603.954} C_VEL
LIN {X 0,Y 552.332,Z 356.187,A -85,B 0,C 180,E1 26600.784,E2 26600.784} C_VEL
LIN {X 0,Y 552.268,Z 356.186,A -85,B 0,C 180,E1 26597.661,E2 26597.661} C_VEL
LIN {X 0,Y 552.29,Z 356.189,A -85,B 0,C 180,E1 26594.33,E2 26594.33} C_VEL
LIN {X 0,Y 552.287,Z 356.173,A -85,B 0,C 180,E1 26591.221,E2 26591.221} C_VEL
LIN {X 0,Y 552.273,Z 356.186,A -85,B 0,C 180,E1 26587.991,E2 26587.991} C_VEL
LIN {X 0,Y 552.299,Z 356.424,A -85,B 0,C 180,E1 26585.626,E2 26585.626} C_VEL
LIN {X 0,Y 556.017,Z 369.918,A -85,B 0,C 180,E1 26583.631,E2 26583.631} C_VEL
LIN {X 0,Y 555.398,Z 395.075,A -85,B 0,C 180,E1 26580.523,E2 26580.523} C_VEL
LIN {X 0,Y 558.7,Z 407.684,A -85,B 0,C 180,E1 26580.128,E2 26580.128} C_VEL
LIN {X 0,Y 557.343,Z 642.619,A -85,B 0,C 180,E1 26576.833,E2 26576.833} C_VEL
LIN {X 0,Y 557.07,Z 663.168,A -85,B 0,C 180,E1 26576.448,E2 26576.448} C_VEL
LIN {X 0,Y 556.68,Z 682.661,A -85,B 0,C 180,E1 26575.913,E2 26575.913} C_VEL
LIN {X 0,Y 556.159,Z 703.996,A -85,B 0,C 180,E1 26575.104,E2 26575.104} C_VEL
LIN {X 0,Y 555.652,Z 722.288,A -85,B 0,C 180,E1 26574.221,E2 26574.221} C_VEL
LIN {X 0,Y 555.049,Z 741.399,A -85,B 0,C 180,E1 26573.086,E2 26573.086} C_VEL
LIN {X 0,Y 554.467,Z 758.485,A -85,B 0,C 180,E1 26571.862,E2 26571.862} C_VEL
LIN {X 0,Y 553.93,Z 774.909,A -85,B 0,C 180,E1 26570.476,E2 26570.476} C_VEL
LIN {X 0,Y 553.407,Z 790.453,A -85,B 0,C 180,E1 26568.923,E2 26568.923} C_VEL
LIN {X 0,Y 552.973,Z 804.784,A -85,B 0,C 180,E1 26567.249,E2 26567.249} C_VEL
LIN {X 0,Y 552.583,Z 818.618,A -85,B 0,C 180,E1 26565.327,E2 26565.327} C_VEL
LIN {X 0,Y 552.336,Z 829.712,A -85,B 0,C 180,E1 26563.504,E2 26563.504} C_VEL
LIN {X 0,Y 552.136,Z 839.849,A -85,B 0,C 180,E1 26561.49,E2 26561.49} C_VEL
LIN {X 0,Y 552.023,Z 847.669,A -85,B 0,C 180,E1 26559.592,E2 26559.592} C_VEL
LIN {X 0,Y 551.956,Z 854.531,A -85,B 0,C 180,E1 26557.494,E2 26557.494} C_VEL
LIN {X 0,Y 551.92,Z 859.539,A -85,B 0,C 180,E1 26555.405,E2 26555.405} C_VEL
LIN {X 0,Y 551.91,Z 862.964,A -85,B 0,C 180,E1 26553.323,E2 26553.323} C_VEL
LIN {X 0,Y 551.91,Z 864.733,A -85,B 0,C 180,E1 26551.142,E2 26551.142} C_VEL
LIN {X 0,Y 551.91,Z 864.82,A -85,B 0,C 180,E1 26549.17,E2 26549.17} C_VEL
LIN {X 0,Y 551.915,Z 863.414,A -85,B 0,C 180,E1 26547.092,E2 26547.092} C_VEL
LIN {X 0,Y 551.924,Z 860.154,A -85,B 0,C 180,E1 26544.907,E2 26544.907} C_VEL
LIN {X 0,Y 551.951,Z 855.679,A -85,B 0,C 180,E1 26542.924,E2 26542.924} C_VEL
LIN {X 0,Y 552.015,Z 848.856,A -85,B 0,C 180,E1 26540.723,E2 26540.723} C_VEL
LIN {X 0,Y 552.106,Z 841.242,A -85,B 0,C 180,E1 26538.827,E2 26538.827} C_VEL
LIN {X 0,Y 552.295,Z 831.444,A -85,B 0,C 180,E1 26536.815,E2 26536.815} C_VEL
LIN {X 0,Y 552.547,Z 820.074,A -85,B 0,C 180,E1 26534.896,E2 26534.896} C_VEL
LIN {X 0,Y 552.868,Z 808.113,A -85,B 0,C 180,E1 26533.181,E2 26533.181} C_VEL
LIN {X 0,Y 553.317,Z 793.284,A -85,B 0,C 180,E1 26531.385,E2 26531.385} C_VEL
LIN {X 0,Y 553.766,Z 779.26,A -85,B 0,C 180,E1 26529.937,E2 26529.937} C_VEL
LIN {X 0,Y 554.369,Z 762.017,A -85,B 0,C 180,E1 26528.412,E2 26528.412} C_VEL
LIN {X 0,Y 554.926,Z 744.907,A -85,B 0,C 180,E1 26527.153,E2 26527.153} C_VEL
LIN {X 0,Y 555.496,Z 727.175,A -85,B 0,C 180,E1 26526.044,E2 26526.044} C_VEL
LIN {X 0,Y 556.049,Z 707.72,A -85,B 0,C 180,E1 26525.061,E2 26525.061} C_VEL
LIN {X 0,Y 556.517,Z 690.034,A -85,B 0,C 180,E1 26524.343,E2 26524.343} C_VEL
LIN {X 0,Y 556.966,Z 669.188,A -85,B 0,C 180,E1 26523.693,E2 26523.693} C_VEL
LIN {X 0,Y 557.261,Z 649.129,A -85,B 0,C 180,E1 26523.274,E2 26523.274} C_VEL
LIN {X 0,Y 558.664,Z 413.989,A -85,B 0,C 180,E1 26519.962,E2 26519.962} C_VEL
LIN {X 0,Y 558.494,Z 406.168,A -85,B 0,C 180,E1 26519.838,E2 26519.838} C_VEL
LIN {X 0,Y 555.367,Z 394.821,A -85,B 0,C 180,E1 26519.46,E2 26519.46} C_VEL
LIN {X 0,Y 556.009,Z 369.208,A -85,B 0,C 180,E1 26516.279,E2 26516.279} C_VEL
LIN {X 0,Y 552.278,Z 356.279,A -85,B 0,C 180,E1 26514.326,E2 26514.326} C_VEL
LIN {X 0,Y 552.325,Z 356.187,A -85,B 0,C 180,E1 26511.118,E2 26511.118} C_VEL
LIN {X 0,Y 552.267,Z 356.179,A -85,B 0,C 180,E1 26508.084,E2 26508.084} C_VEL
LIN {X 0,Y 552.295,Z 356.187,A -85,B 0,C 180,E1 26504.77,E2 26504.77} C_VEL
LIN {X 0,Y 552.277,Z 356.185,A -85,B 0,C 180,E1 26501.766,E2 26501.766} C_VEL
LIN {X 0,Y 552.271,Z 356.183,A -85,B 0,C 180,E1 26498.381,E2 26498.381} C_VEL
LIN {X 0,Y 552.315,Z 356.187,A -85,B 0,C 180,E1 26495.272,E2 26495.272} C_VEL
LIN {X 0,Y 552.265,Z 356.186,A -85,B 0,C 180,E1 26492.04,E2 26492.04} C_VEL
LIN {X 0,Y 552.331,Z 356.177,A -85,B 0,C 180,E1 26488.82,E2 26488.82} C_VEL
LIN {X 0,Y 552.268,Z 356.186,A -85,B 0,C 180,E1 26485.633,E2 26485.633} C_VEL
LIN {X 0,Y 552.278,Z 356.178,A -85,B 0,C 180,E1 26482.236,E2 26482.236} C_VEL
LIN {X 0,Y 552.298,Z 356.183,A -85,B 0,C 180,E1 26479.131,E2 26479.131} C_VEL
LIN {X 0,Y 552.264,Z 356.183,A -85,B 0,C 180,E1 26475.869,E2 26475.869} C_VEL
LIN {X 0,Y 552.33,Z 356.176,A -85,B 0,C 180,E1 26472.763,E2 26472.763} C_VEL
LIN {X 0,Y 552.262,Z 356.187,A -85,B 0,C 180,E1 26469.592,E2 26469.592} C_VEL
LIN {X 0,Y 552.313,Z 356.175,A -85,B 0,C 180,E1 26466.344,E2 26466.344} C_VEL
LIN {X 0,Y 552.269,Z 356.186,A -85,B 0,C 180,E1 26463.222,E2 26463.222} C_VEL
LIN {X 0,Y 552.269,Z 356.179,A -85,B 0,C 180,E1 26459.797,E2 26459.797} C_VEL
LIN {X 0,Y 552.306,Z 356.179,A -85,B 0,C 180,E1 26456.684,E2 26456.684} C_VEL
LIN {X 0,Y 552.261,Z 356.186,A -85,B 0,C 180,E1 26453.456,E2 26453.456} C_VEL
LIN {X 0,Y 552.33,Z 356.173,A -85,B 0,C 180,E1 26450.313,E2 26450.313} C_VEL
LIN {X 0,Y 552.262,Z 356.187,A -85,B 0,C 180,E1 26447.139,E2 26447.139} C_VEL
LIN {X 0,Y 552.306,Z 356.176,A -85,B 0,C 180,E1 26443.926,E2 26443.926} C_VEL
LIN {X 0,Y 552.267,Z 356.184,A -85,B 0,C 180,E1 26440.877,E2 26440.877} C_VEL
LIN {X 0,Y 552.269,Z 356.182,A -85,B 0,C 180,E1 26437.414,E2 26437.414} C_VEL
LIN {X 0,Y 552.312,Z 356.181,A -85,B 0,C 180,E1 26434.255,E2 26434.255} C_VEL
LIN {X 0,Y 552.267,Z 356.188,A -85,B 0,C 180,E1 26432.734,E2 26432.734} C_VEL
LIN {X 0,Y 551.304,Z 356.316,A -85,B 0,C 180,E1 26431.935,E2 26431.935} C_VEL
LIN {X 0,Y 544.77,Z 357.127,A -85,B 0,C 180,E1 26429.632,E2 26429.632} C_VEL
LIN {X 0,Y 544.323,Z 357.177,A -85,B 0,C 180,E1 26429.105,E2 26429.105} C_VEL
LIN {X 0,Y 544.391,Z 357.177,A -85,B 0,C 180,E1 26425.925,E2 26425.925} C_VEL
LIN {X 0,Y 544.324,Z 357.176,A -85,B 0,C 180,E1 26422.688,E2 26422.688} C_VEL
LIN {X 0,Y 544.346,Z 357.177,A -85,B 0,C 180,E1 26419.339,E2 26419.339} C_VEL
LIN {X 0,Y 544.335,Z 357.177,A -85,B 0,C 180,E1 26416.329,E2 26416.329} C_VEL
LIN {X 0,Y 544.326,Z 357.178,A -85,B 0,C 180,E1 26412.958,E2 26412.958} C_VEL
LIN {X 0,Y 544.373,Z 357.176,A -85,B 0,C 180,E1 26409.86,E2 26409.86} C_VEL
LIN {X 0,Y 544.319,Z 357.178,A -85,B 0,C 180,E1 26406.622,E2 26406.622} C_VEL
LIN {X 0,Y 544.387,Z 357.177,A -85,B 0,C 180,E1 26403.435,E2 26403.435} C_VEL
LIN {X 0,Y 544.327,Z 357.177,A -85,B 0,C 180,E1 26400.218,E2 26400.218} C_VEL
LIN {X 0,Y 544.327,Z 357.178,A -85,B 0,C 180,E1 26396.745,E2 26396.745} C_VEL
LIN {X 0,Y 544.371,Z 357.178,A -85,B 0,C 180,E1 26393.598,E2 26393.598} C_VEL
LIN {X 0,Y 544.318,Z 357.177,A -85,B 0,C 180,E1 26390.426,E2 26390.426} C_VEL
LIN {X 0,Y 544.385,Z 357.177,A -85,B 0,C 180,E1 26387.199,E2 26387.199} C_VEL
LIN {X 0,Y 544.321,Z 357.178,A -85,B 0,C 180,E1 26384.032,E2 26384.032} C_VEL
LIN {X 0,Y 544.341,Z 357.178,A -85,B 0,C 180,E1 26380.691,E2 26380.691} C_VEL
LIN {X 0,Y 544.34,Z 357.179,A -85,B 0,C 180,E1 26377.599,E2 26377.599} C_VEL
LIN {X 0,Y 544.322,Z 357.177,A -85,B 0,C 180,E1 26374.319,E2 26374.319} C_VEL
LIN {X 0,Y 544.389,Z 357.177,A -85,B 0,C 180,E1 26371.052,E2 26371.052} C_VEL
LIN {X 0,Y 544.317,Z 357.178,A -85,B 0,C 180,E1 26367.895,E2 26367.895} C_VEL
LIN {X 0,Y 544.36,Z 357.178,A -85,B 0,C 180,E1 26364.625,E2 26364.625} C_VEL
LIN {X 0,Y 544.325,Z 357.179,A -85,B 0,C 180,E1 26361.55,E2 26361.55} C_VEL
LIN {X 0,Y 544.326,Z 357.177,A -85,B 0,C 180,E1 26358.128,E2 26358.128} C_VEL
LIN {X 0,Y 544.368,Z 357.178,A -85,B 0,C 180,E1 26354.991,E2 26354.991} C_VEL
LIN {X 0,Y 544.318,Z 357.178,A -85,B 0,C 180,E1 26351.719,E2 26351.719} C_VEL
LIN {X 0,Y 544.372,Z 357.177,A -85,B 0,C 180,E1 26348.449,E2 26348.449} C_VEL
LIN {X 0,Y 544.323,Z 357.178,A -85,B 0,C 180,E1 26345.357,E2 26345.357} C_VEL
LIN {X 0,Y 544.333,Z 357.177,A -85,B 0,C 180,E1 26341.951,E2 26341.951} C_VEL
LIN {X 0,Y 544.347,Z 357.177,A -85,B 0,C 180,E1 26338.927,E2 26338.927} C_VEL
LIN {X 0,Y 544.324,Z 357.178,A -85,B 0,C 180,E1 26335.674,E2 26335.674} C_VEL
LIN {X 0,Y 544.39,Z 357.177,A -85,B 0,C 180,E1 26332.428,E2 26332.428} C_VEL
LIN {X 0,Y 544.319,Z 357.177,A -85,B 0,C 180,E1 26329.301,E2 26329.301} C_VEL
LIN {X 0,Y 544.369,Z 357.177,A -85,B 0,C 180,E1 26326.032,E2 26326.032} C_VEL
LIN {X 0,Y 544.331,Z 357.178,A -85,B 0,C 180,E1 26322.871,E2 26322.871} C_VEL
LIN {X 0,Y 544.326,Z 357.177,A -85,B 0,C 180,E1 26319.452,E2 26319.452} C_VEL
LIN {X 0,Y 544.366,Z 357.177,A -85,B 0,C 180,E1 26316.38,E2 26316.38} C_VEL
LIN {X 0,Y 544.322,Z 357.177,A -85,B 0,C 180,E1 26313.113,E2 26313.113} C_VEL
LIN {X 0,Y 544.38,Z 357.176,A -85,B 0,C 180,E1 26309.843,E2 26309.843} C_VEL
LIN {X 0,Y 544.326,Z 357.177,A -85,B 0,C 180,E1 26306.739,E2 26306.739} C_VEL
LIN {X 0,Y 544.334,Z 357.17,A -85,B 0,C 180,E1 26303.307,E2 26303.307} C_VEL
LIN {X 0,Y 544.362,Z 357.177,A -85,B 0,C 180,E1 26300.19,E2 26300.19} C_VEL
LIN {X 0,Y 544.322,Z 357.163,A -85,B 0,C 180,E1 26296.976,E2 26296.976} C_VEL
LIN {X 0,Y 544.397,Z 357.175,A -85,B 0,C 180,E1 26293.808,E2 26293.808} C_VEL
LIN {X 0,Y 544.323,Z 357.169,A -85,B 0,C 180,E1 26290.579,E2 26290.579} C_VEL
LIN {X 0,Y 544.355,Z 357.175,A -85,B 0,C 180,E1 26287.276,E2 26287.276} C_VEL
LIN {X 0,Y 544.34,Z 357.176,A -85,B 0,C 180,E1 26284.159,E2 26284.159} C_VEL
LIN {X 0,Y 544.327,Z 357.167,A -85,B 0,C 180,E1 26280.837,E2 26280.837} C_VEL
LIN {X 0,Y 544.379,Z 357.176,A -85,B 0,C 180,E1 26277.68,E2 26277.68} C_VEL
LIN {X 0,Y 544.324,Z 357.166,A -85,B 0,C 180,E1 26274.409,E2 26274.409} C_VEL
LIN {X 0,Y 544.374,Z 357.175,A -85,B 0,C 180,E1 26271.16,E2 26271.16} C_VEL
LIN {X 0,Y 544.332,Z 357.175,A -85,B 0,C 180,E1 26268.017,E2 26268.017} C_VEL
LIN {X 0,Y 544.329,Z 357.171,A -85,B 0,C 180,E1 26264.55,E2 26264.55} C_VEL
LIN {X 0,Y 544.388,Z 357.176,A -85,B 0,C 180,E1 26261.359,E2 26261.359} C_VEL
LIN {X 0,Y 544.325,Z 357.165,A -85,B 0,C 180,E1 26258.103,E2 26258.103} C_VEL
LIN {X 0,Y 544.374,Z 357.174,A -85,B 0,C 180,E1 26254.887,E2 26254.887} C_VEL
LIN {X 0,Y 544.336,Z 357.164,A -85,B 0,C 180,E1 26251.709,E2 26251.709} C_VEL
LIN {X 0,Y 544.331,Z 357.175,A -85,B 0,C 180,E1 26248.26,E2 26248.26} C_VEL
LIN {X 0,Y 544.401,Z 357.174,A -85,B 0,C 180,E1 26244.996,E2 26244.996} C_VEL
LIN {X 0,Y 544.329,Z 357.171,A -85,B 0,C 180,E1 26241.753,E2 26241.753} C_VEL
LIN {X 0,Y 544.358,Z 357.173,A -85,B 0,C 180,E1 26238.463,E2 26238.463} C_VEL
LIN {X 0,Y 544.35,Z 357.176,A -85,B 0,C 180,E1 26235.302,E2 26235.302} C_VEL
LIN {X 0,Y 544.328,Z 357.168,A -85,B 0,C 180,E1 26231.93,E2 26231.93} C_VEL
LIN {X 0,Y 544.4,Z 357.176,A -85,B 0,C 180,E1 26228.685,E2 26228.685} C_VEL
LIN {X 0,Y 544.374,Z 357.402,A -85,B 0,C 180,E1 26226.061,E2 26226.061} C_VEL
LIN {X 0,Y 548.573,Z 372.146,A -85,B 0,C 180,E1 26223.829,E2 26223.829} C_VEL
LIN {X 0,Y 548.014,Z 395.237,A -85,B 0,C 180,E1 26220.972,E2 26220.972} C_VEL
LIN {X 0,Y 551.769,Z 409.536,A -85,B 0,C 180,E1 26220.519,E2 26220.519} C_VEL
LIN {X 0,Y 550.182,Z 644.028,A -85,B 0,C 180,E1 26217.187,E2 26217.187} C_VEL
LIN {X 0,Y 549.88,Z 663.721,A -85,B 0,C 180,E1 26216.807,E2 26216.807} C_VEL
LIN {X 0,Y 549.445,Z 682.888,A -85,B 0,C 180,E1 26216.273,E2 26216.273} C_VEL
LIN {X 0,Y 548.857,Z 703.981,A -85,B 0,C 180,E1 26215.462,E2 26215.462} C_VEL
LIN {X 0,Y 548.263,Z 722.271,A -85,B 0,C 180,E1 26214.569,E2 26214.569} C_VEL
LIN {X 0,Y 547.542,Z 741.961,A -85,B 0,C 180,E1 26213.382,E2 26213.382} C_VEL
LIN {X 0,Y 546.934,Z 757.767,A -85,B 0,C 180,E1 26212.235,E2 26212.235} C_VEL
LIN {X 0,Y 546.286,Z 774.681,A -85,B 0,C 180,E1 26210.797,E2 26210.797} C_VEL
LIN {X 0,Y 545.66,Z 790.667,A -85,B 0,C 180,E1 26209.177,E2 26209.177} C_VEL
LIN {X 0,Y 545.155,Z 804.846,A -85,B 0,C 180,E1 26207.497,E2 26207.497} C_VEL
LIN {X 0,Y 544.727,Z 817.975,A -85,B 0,C 180,E1 26205.653,E2 26205.653} C_VEL
LIN {X 0,Y 544.421,Z 829.103,A -85,B 0,C 180,E1 26203.812,E2 26203.812} C_VEL
